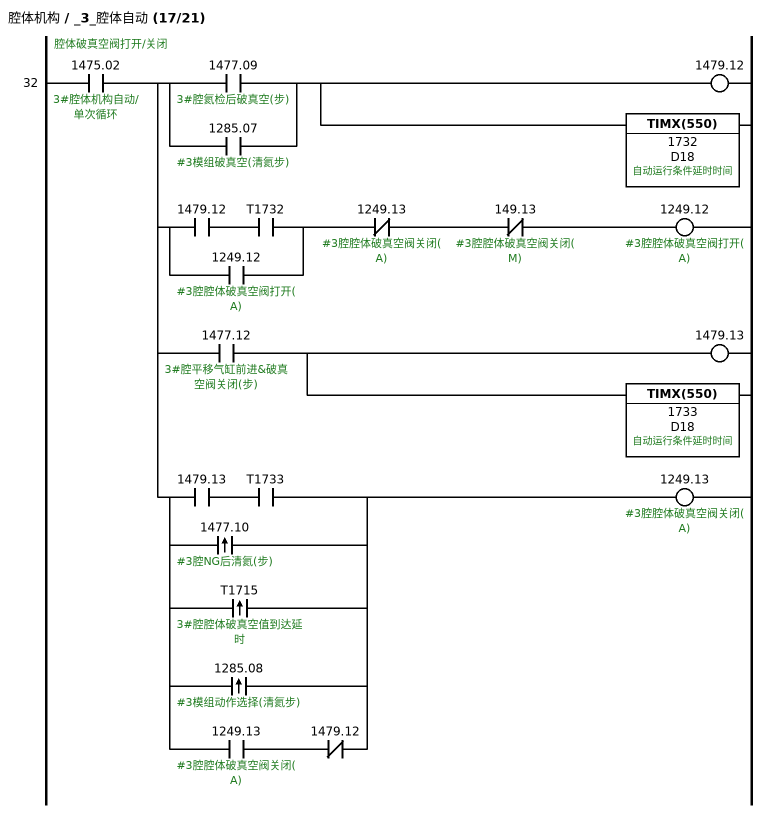
; [picture p336: 腔体机构 / _3_腔体自动, rungs 32-32]
; rung 32: 腔体破真空阀打开/关闭
LD 1475.02  ; 3#腔体机构自动/单次循环
OUT TR0
LD 1477.09  ; 3#腔氦检后破真空(步)
OR 1285.07  ; #3模组破真空(清氦步)
ANDLD
OUT 1479.12
TIMX(550) 1732 D18  ; 自动运行条件延时时间
LD TR0
LD 1479.12
AND T1732
OR 1249.12  ; #3腔腔体破真空阀打开(A)
ANDLD
ANDNOT 1249.13  ; #3腔腔体破真空阀关闭(A)
ANDNOT 149.13  ; #3腔腔体破真空阀关闭(M)
OUT 1249.12  ; #3腔腔体破真空阀打开(A)
LD TR0
AND 1477.12  ; 3#腔平移气缸前进&破真空阀关闭(步)
OUT 1479.13
TIMX(550) 1733 D18  ; 自动运行条件延时时间
LD TR0
LD 1479.13
AND T1733
@OR 1477.10  ; #3腔NG后清氦(步)
@OR T1715  ; 3#腔腔体破真空值到达延时
@OR 1285.08  ; #3模组动作选择(清氦步)
LD 1249.13  ; #3腔腔体破真空阀关闭(A)
ANDNOT 1479.12
ORLD
ANDLD
OUT 1249.13  ; #3腔腔体破真空阀关闭(A)

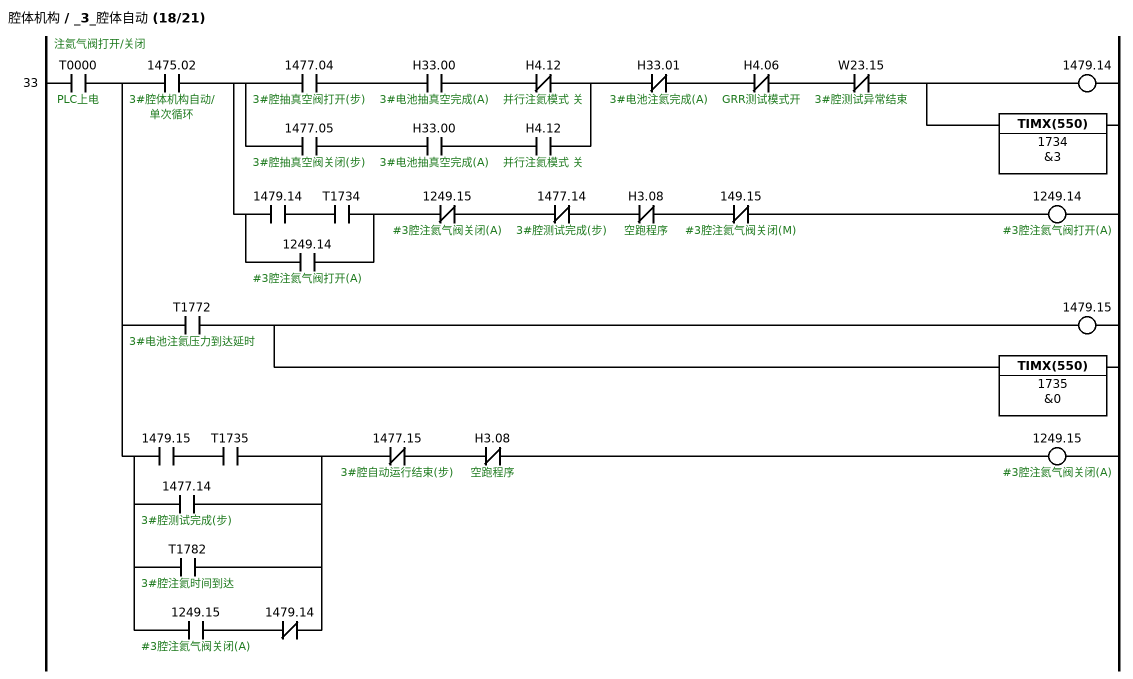
; rung 33: 注氦气阀打开/关闭
LD T0000  ; PLC上电
OUT TR0
AND 1475.02  ; 3#腔体机构自动/单次循环
OUT TR1
LD 1477.04  ; 3#腔抽真空阀打开(步)
AND H33.00  ; 3#电池抽真空完成(A)
ANDNOT H4.12  ; 并行注氦模式 关
LD 1477.05  ; 3#腔抽真空阀关闭(步)
AND H33.00  ; 3#电池抽真空完成(A)
AND H4.12  ; 并行注氦模式 关
ORLD
ANDLD
ANDNOT H33.01  ; 3#电池注氦完成(A)
ANDNOT H4.06  ; GRR测试模式开
ANDNOT W23.15  ; 3#腔测试异常结束
OUT 1479.14
TIMX(550) 1734 &3
LD TR1
LD 1479.14
AND T1734
OR 1249.14  ; #3腔注氦气阀打开(A)
ANDLD
ANDNOT 1249.15  ; #3腔注氦气阀关闭(A)
ANDNOT 1477.14  ; 3#腔测试完成(步)
ANDNOT H3.08  ; 空跑程序
ANDNOT 149.15  ; #3腔注氦气阀关闭(M)
OUT 1249.14  ; #3腔注氦气阀打开(A)
LD TR0
AND T1772  ; 3#电池注氦压力到达延时
OUT 1479.15
TIMX(550) 1735 &0
LD TR0
LD 1479.15
AND T1735
OR 1477.14  ; 3#腔测试完成(步)
OR T1782  ; 3#腔注氦时间到达
LD 1249.15  ; #3腔注氦气阀关闭(A)
ANDNOT 1479.14
ORLD
ANDLD
ANDNOT 1477.15  ; 3#腔自动运行结束(步)
ANDNOT H3.08  ; 空跑程序
OUT 1249.15  ; #3腔注氦气阀关闭(A)

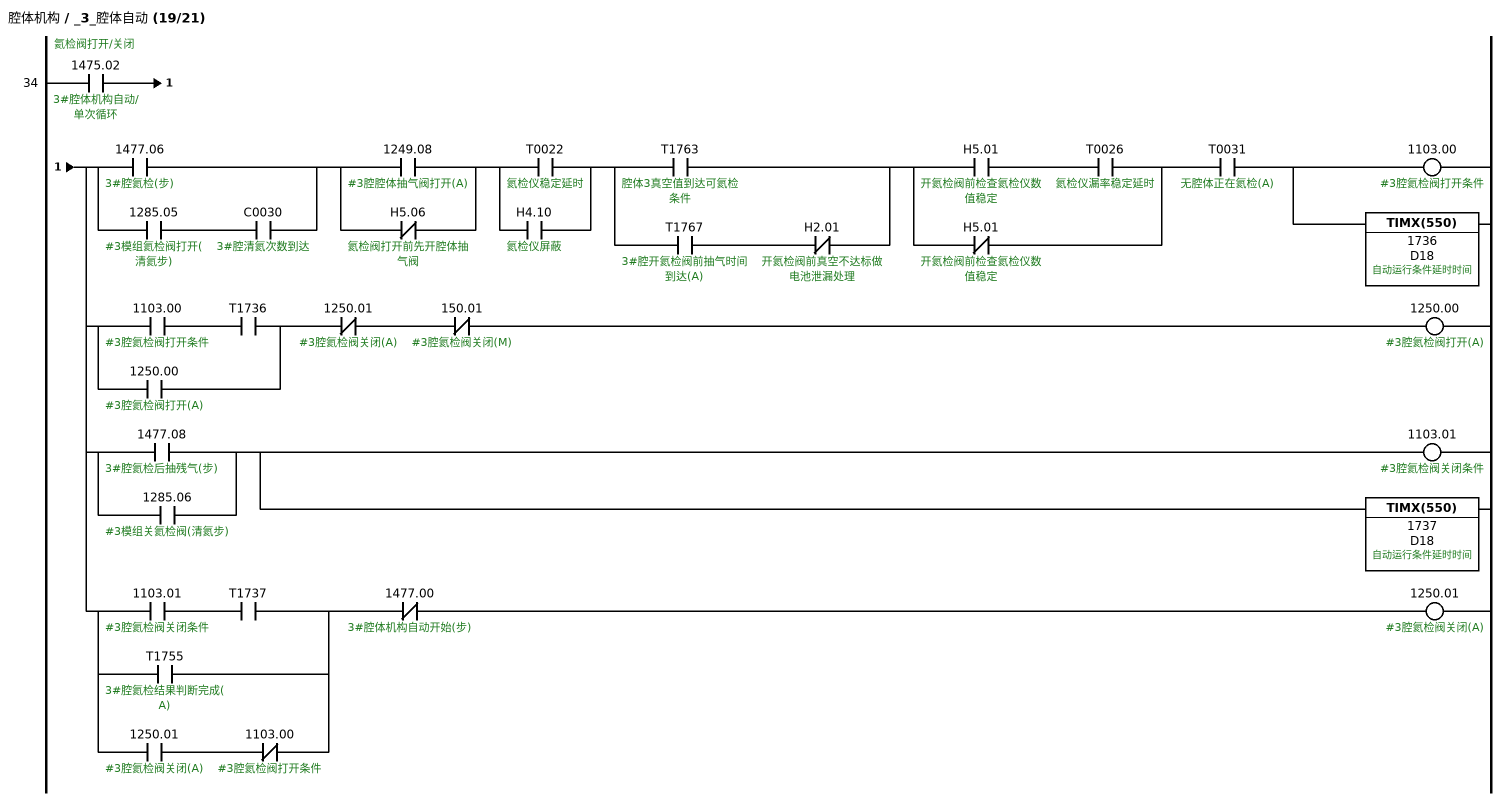
; rung 34: 氦检阀打开/关闭
LD 1475.02  ; 3#腔体机构自动/单次循环
OUT TR0
LD 1477.06  ; 3#腔氦检(步)
LD 1285.05  ; #3模组氦检阀打开(清氦步)
AND C0030  ; 3#腔清氦次数到达
ORLD
ANDLD
LD 1249.08  ; #3腔腔体抽气阀打开(A)
ORNOT H5.06  ; 氦检阀打开前先开腔体抽气阀
ANDLD
LD T0022  ; 氦检仪稳定延时
OR H4.10  ; 氦检仪屏蔽
ANDLD
LD T1763  ; 腔体3真空值到达可氦检条件
LD T1767  ; 3#腔开氦检阀前抽气时间到达(A)
ANDNOT H2.01  ; 开氦检阀前真空不达标做电池泄漏处理
ORLD
ANDLD
LD H5.01  ; 开氦检阀前检查氦检仪数值稳定
AND T0026  ; 氦检仪漏率稳定延时
ORNOT H5.01  ; 开氦检阀前检查氦检仪数值稳定
ANDLD
AND T0031  ; 无腔体正在氦检(A)
OUT 1103.00  ; #3腔氦检阀打开条件
TIMX(550) 1736 D18  ; 自动运行条件延时时间
LD TR0
LD 1103.00  ; #3腔氦检阀打开条件
AND T1736
OR 1250.00  ; #3腔氦检阀打开(A)
ANDLD
ANDNOT 1250.01  ; #3腔氦检阀关闭(A)
ANDNOT 150.01  ; #3腔氦检阀关闭(M)
OUT 1250.00  ; #3腔氦检阀打开(A)
LD TR0
LD 1477.08  ; 3#腔氦检后抽残气(步)
OR 1285.06  ; #3模组关氦检阀(清氦步)
ANDLD
OUT 1103.01  ; #3腔氦检阀关闭条件
TIMX(550) 1737 D18  ; 自动运行条件延时时间
LD TR0
LD 1103.01  ; #3腔氦检阀关闭条件
AND T1737
OR T1755  ; 3#腔氦检结果判断完成(A)
LD 1250.01  ; #3腔氦检阀关闭(A)
ANDNOT 1103.00  ; #3腔氦检阀打开条件
ORLD
ANDLD
ANDNOT 1477.00  ; 3#腔体机构自动开始(步)
OUT 1250.01  ; #3腔氦检阀关闭(A)

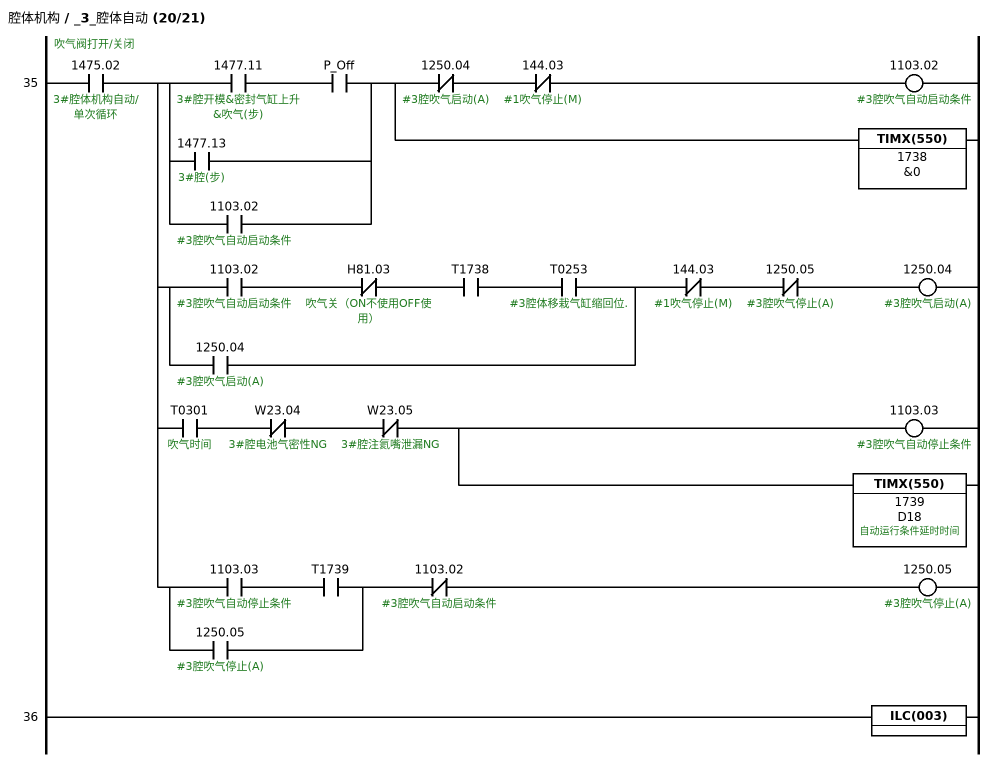
; rung 35: 吹气阀打开/关闭
LD 1475.02  ; 3#腔体机构自动/单次循环
OUT TR0
LD 1477.11  ; 3#腔开模&密封气缸上升&吹气(步)
AND P_Off
OR 1477.13  ; 3#腔(步)
OR 1103.02  ; #3腔吹气自动启动条件
ANDLD
OUT TR1
ANDNOT 1250.04  ; #3腔吹气启动(A)
ANDNOT 144.03  ; #1吹气停止(M)
OUT 1103.02  ; #3腔吹气自动启动条件
LD TR1
TIMX(550) 1738 &0
LD TR0
LD 1103.02  ; #3腔吹气自动启动条件
ANDNOT H81.03  ; 吹气关（ON不使用OFF使用）
AND T1738
AND T0253  ; #3腔体移栽气缸缩回位.
OR 1250.04  ; #3腔吹气启动(A)
ANDLD
ANDNOT 144.03  ; #1吹气停止(M)
ANDNOT 1250.05  ; #3腔吹气停止(A)
OUT 1250.04  ; #3腔吹气启动(A)
LD TR0
AND T0301  ; 吹气时间
ANDNOT W23.04  ; 3#腔电池气密性NG
ANDNOT W23.05  ; 3#腔注氦嘴泄漏NG
OUT 1103.03  ; #3腔吹气自动停止条件
TIMX(550) 1739 D18  ; 自动运行条件延时时间
LD TR0
LD 1103.03  ; #3腔吹气自动停止条件
AND T1739
OR 1250.05  ; #3腔吹气停止(A)
ANDLD
ANDNOT 1103.02  ; #3腔吹气自动启动条件
OUT 1250.05  ; #3腔吹气停止(A)
; rung 36
ILC(003)

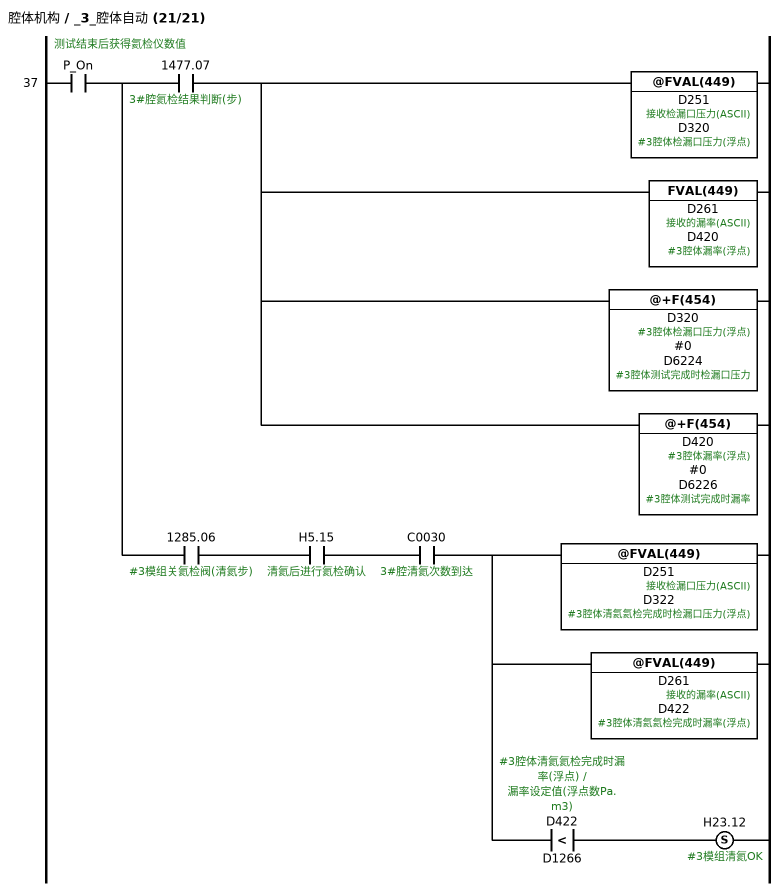
; rung 37: 测试结束后获得氦检仪数值
LD P_On
OUT TR0
AND 1477.07  ; 3#腔氦检结果判断(步)
@FVAL(449) D251 D320  ; 接收检漏口压力(ASCII), #3腔体检漏口压力(浮点)
FVAL(449) D261 D420  ; 接收的漏率(ASCII), #3腔体漏率(浮点)
@+F(454) D320 #0 D6224  ; #3腔体检漏口压力(浮点), #3腔体测试完成时检漏口压力
@+F(454) D420 #0 D6226  ; #3腔体漏率(浮点), #3腔体测试完成时漏率
LD TR0
AND 1285.06  ; #3模组关氦检阀(清氦步)
AND H5.15  ; 清氦后进行氦检确认
AND C0030  ; 3#腔清氦次数到达
@FVAL(449) D251 D322  ; 接收检漏口压力(ASCII), #3腔体清氦氦检完成时检漏口压力(浮点)
@FVAL(449) D261 D422  ; 接收的漏率(ASCII), #3腔体清氦氦检完成时漏率(浮点)
AND<F(331) D422 D1266  ; #3腔体清氦氦检完成时漏率(浮点), 漏率设定值(浮点数Pa.m3)
SET H23.12  ; #3模组清氦OK

### Section _4_腔体自动

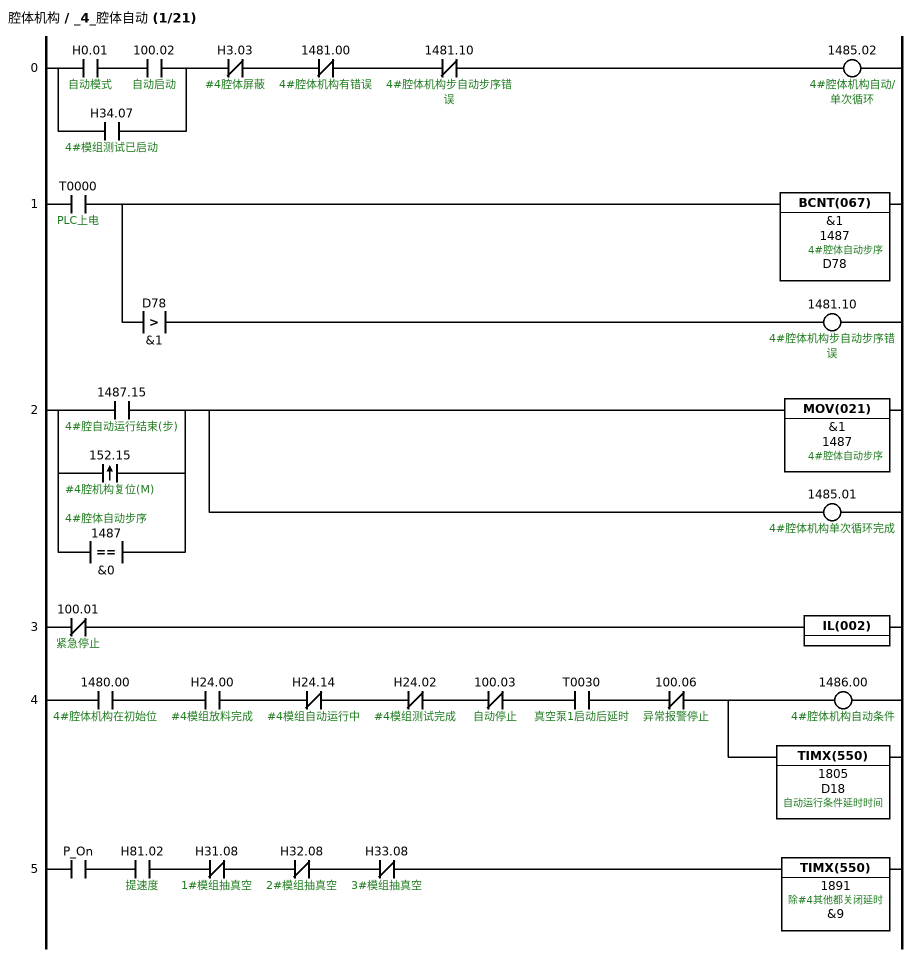
; rung 0
LD H0.01  ; 自动模式
AND 100.02  ; 自动启动
OR H34.07  ; 4#模组测试已启动
ANDNOT H3.03  ; #4腔体屏蔽
ANDNOT 1481.00  ; 4#腔体机构有错误
ANDNOT 1481.10  ; 4#腔体机构步自动步序错误
OUT 1485.02  ; 4#腔体机构自动/单次循环
; rung 1
LD T0000  ; PLC上电
BCNT(067) &1 1487 D78  ; 4#腔体自动步序
AND>(320) D78 &1
OUT 1481.10  ; 4#腔体机构步自动步序错误
; rung 2
LD 1487.15  ; 4#腔自动运行结束(步)
@OR 152.15  ; #4腔机构复位(M)
OR=(300) 1487 &0  ; 4#腔体自动步序
MOV(021) &1 1487  ; 4#腔体自动步序
OUT 1485.01  ; 4#腔体机构单次循环完成
; rung 3
LDNOT 100.01  ; 紧急停止
IL(002)
; rung 4
LD 1480.00  ; 4#腔体机构在初始位
AND H24.00  ; #4模组放料完成
ANDNOT H24.14  ; #4模组自动运行中
ANDNOT H24.02  ; #4模组测试完成
ANDNOT 100.03  ; 自动停止
AND T0030  ; 真空泵1启动后延时
ANDNOT 100.06  ; 异常报警停止
OUT 1486.00  ; 4#腔体机构自动条件
TIMX(550) 1805 D18  ; 自动运行条件延时时间
; rung 5
LD P_On
AND H81.02  ; 提速度
ANDNOT H31.08  ; 1#模组抽真空
ANDNOT H32.08  ; 2#模组抽真空
ANDNOT H33.08  ; 3#模组抽真空
TIMX(550) 1891 &9  ; 除#4其他都关闭延时

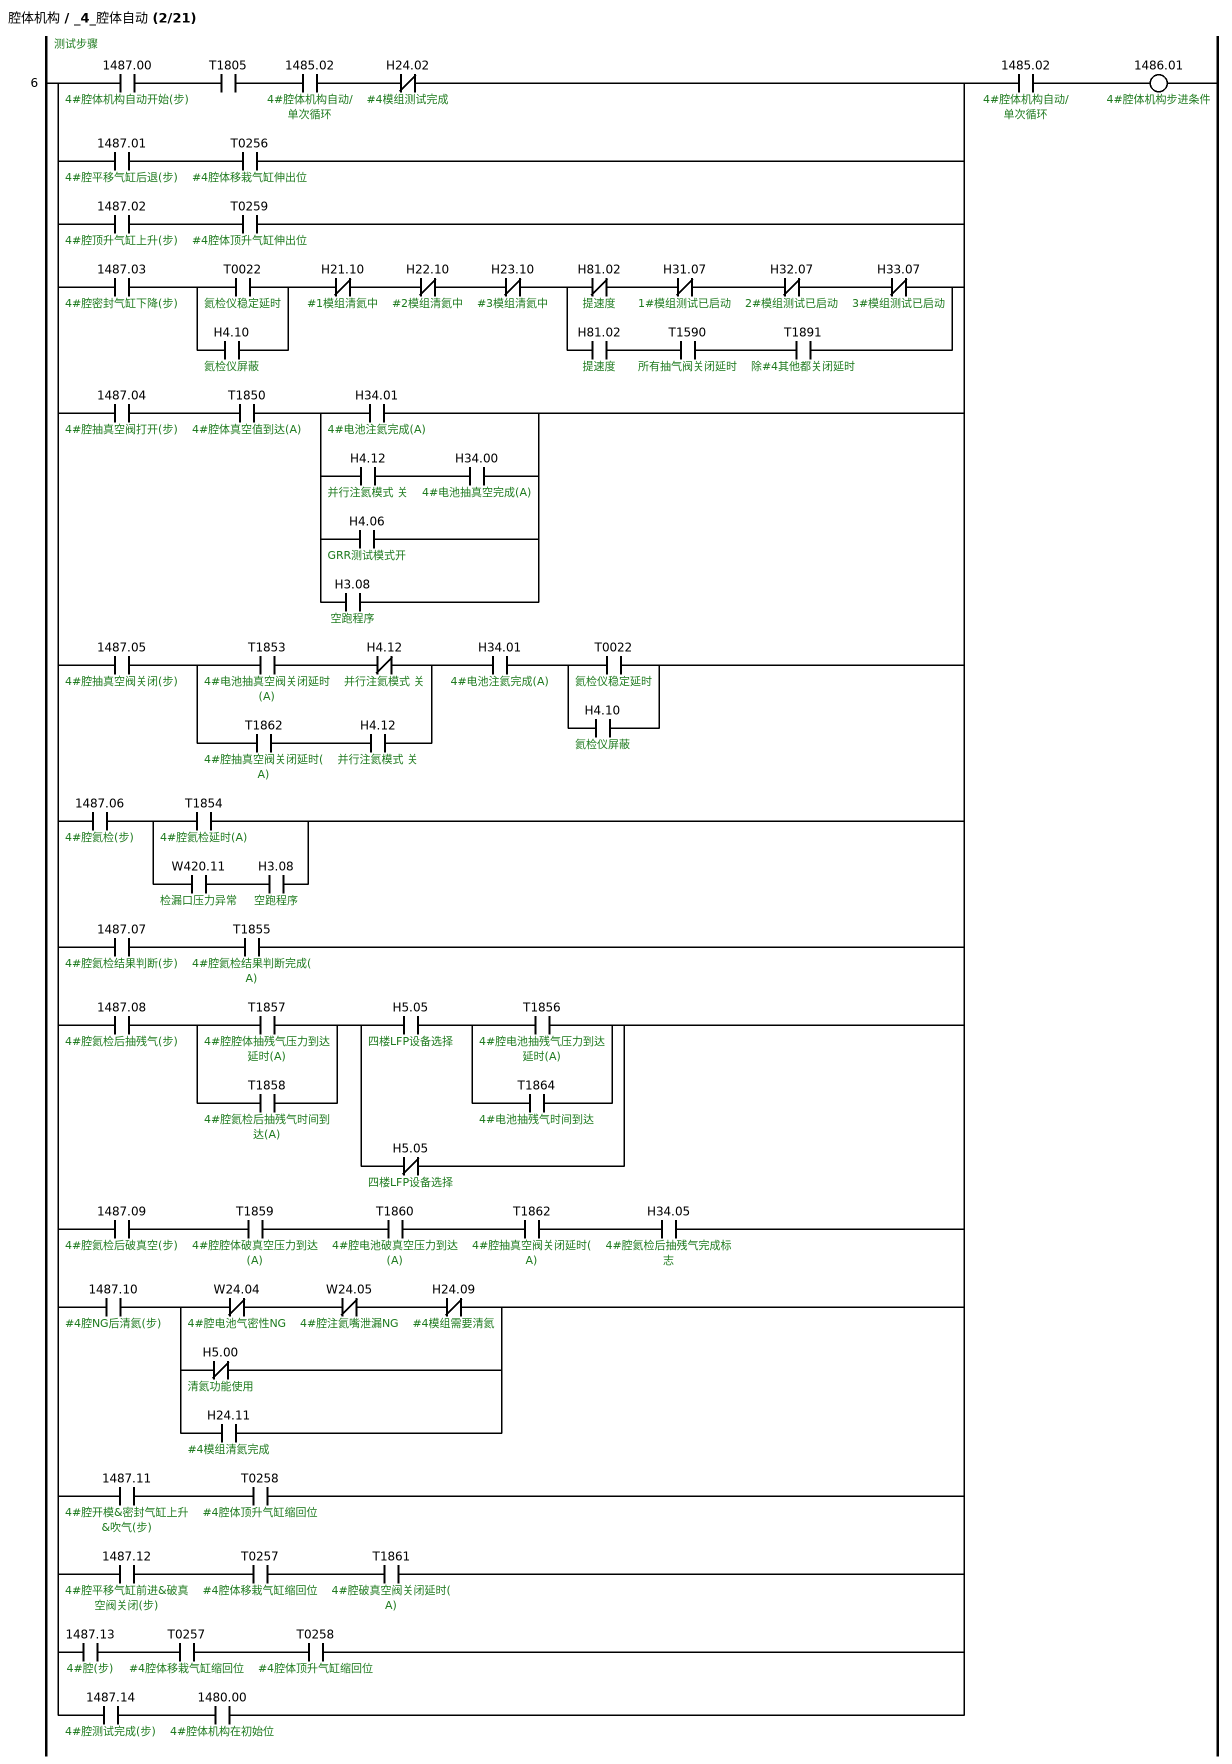
; rung 6: 测试步骤
LD 1487.00  ; 4#腔体机构自动开始(步)
AND T1805
AND 1485.02  ; 4#腔体机构自动/单次循环
ANDNOT H24.02  ; #4模组测试完成
LD 1487.01  ; 4#腔平移气缸后退(步)
AND T0256  ; #4腔体移栽气缸伸出位
ORLD
LD 1487.02  ; 4#腔顶升气缸上升(步)
AND T0259  ; #4腔体顶升气缸伸出位
ORLD
LD 1487.03  ; 4#腔密封气缸下降(步)
LD T0022  ; 氦检仪稳定延时
OR H4.10  ; 氦检仪屏蔽
ANDLD
ANDNOT H21.10  ; #1模组清氦中
ANDNOT H22.10  ; #2模组清氦中
ANDNOT H23.10  ; #3模组清氦中
LDNOT H81.02  ; 提速度
ANDNOT H31.07  ; 1#模组测试已启动
ANDNOT H32.07  ; 2#模组测试已启动
ANDNOT H33.07  ; 3#模组测试已启动
LD H81.02  ; 提速度
AND T1590  ; 所有抽气阀关闭延时
AND T1891  ; 除#4其他都关闭延时
ORLD
ANDLD
ORLD
LD 1487.04  ; 4#腔抽真空阀打开(步)
AND T1850  ; 4#腔体真空值到达(A)
LD H34.01  ; 4#电池注氦完成(A)
LD H4.12  ; 并行注氦模式 关
AND H34.00  ; 4#电池抽真空完成(A)
ORLD
OR H4.06  ; GRR测试模式开
OR H3.08  ; 空跑程序
ANDLD
ORLD
LD 1487.05  ; 4#腔抽真空阀关闭(步)
LD T1853  ; 4#电池抽真空阀关闭延时(A)
ANDNOT H4.12  ; 并行注氦模式 关
LD T1862  ; 4#腔抽真空阀关闭延时(A)
AND H4.12  ; 并行注氦模式 关
ORLD
ANDLD
AND H34.01  ; 4#电池注氦完成(A)
LD T0022  ; 氦检仪稳定延时
OR H4.10  ; 氦检仪屏蔽
ANDLD
ORLD
LD 1487.06  ; 4#腔氦检(步)
LD T1854  ; 4#腔氦检延时(A)
LD W420.11  ; 检漏口压力异常
AND H3.08  ; 空跑程序
ORLD
ANDLD
ORLD
LD 1487.07  ; 4#腔氦检结果判断(步)
AND T1855  ; 4#腔氦检结果判断完成(A)
ORLD
LD 1487.08  ; 4#腔氦检后抽残气(步)
LD T1857  ; 4#腔腔体抽残气压力到达延时(A)
OR T1858  ; 4#腔氦检后抽残气时间到达(A)
ANDLD
LD H5.05  ; 四楼LFP设备选择
LD T1856  ; 4#腔电池抽残气压力到达延时(A)
OR T1864  ; 4#电池抽残气时间到达
ANDLD
ORNOT H5.05  ; 四楼LFP设备选择
ANDLD
ORLD
LD 1487.09  ; 4#腔氦检后破真空(步)
AND T1859  ; 4#腔腔体破真空压力到达(A)
AND T1860  ; 4#腔电池破真空压力到达(A)
AND T1862  ; 4#腔抽真空阀关闭延时(A)
AND H34.05  ; 4#腔氦检后抽残气完成标志
ORLD
LD 1487.10  ; #4腔NG后清氦(步)
LDNOT W24.04  ; 4#腔电池气密性NG
ANDNOT W24.05  ; 4#腔注氦嘴泄漏NG
ANDNOT H24.09  ; #4模组需要清氦
ORNOT H5.00  ; 清氦功能使用
OR H24.11  ; #4模组清氦完成
ANDLD
ORLD
LD 1487.11  ; 4#腔开模&密封气缸上升&吹气(步)
AND T0258  ; #4腔体顶升气缸缩回位
ORLD
LD 1487.12  ; 4#腔平移气缸前进&破真空阀关闭(步)
AND T0257  ; #4腔体移栽气缸缩回位
AND T1861  ; 4#腔破真空阀关闭延时(A)
ORLD
LD 1487.13  ; 4#腔(步)
AND T0257  ; #4腔体移栽气缸缩回位
AND T0258  ; #4腔体顶升气缸缩回位
ORLD
LD 1487.14  ; 4#腔测试完成(步)
AND 1480.00  ; 4#腔体机构在初始位
ORLD
AND 1485.02  ; 4#腔体机构自动/单次循环
OUT 1486.01  ; 4#腔体机构步进条件

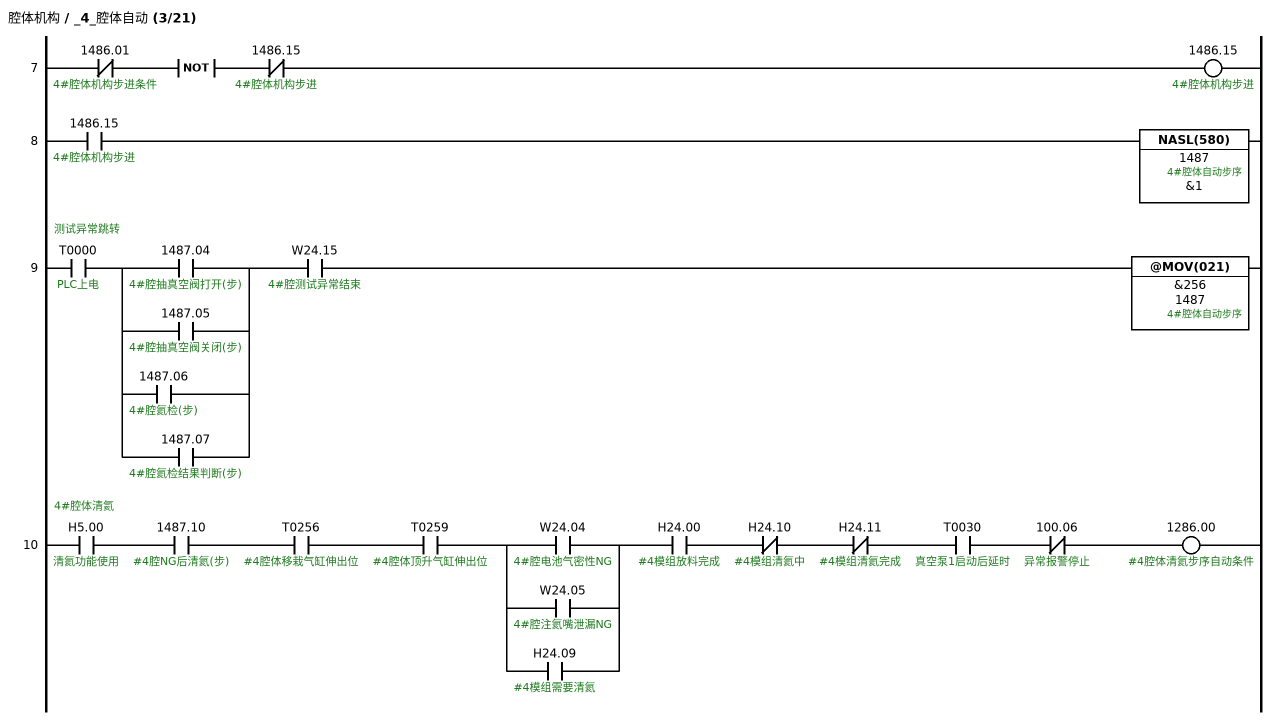
; rung 7
LDNOT 1486.01  ; 4#腔体机构步进条件
NOT(520)
ANDNOT 1486.15  ; 4#腔体机构步进
OUT 1486.15  ; 4#腔体机构步进
; rung 8
LD 1486.15  ; 4#腔体机构步进
NASL(580) 1487 &1  ; 4#腔体自动步序
; rung 9: 测试异常跳转
LD T0000  ; PLC上电
LD 1487.04  ; 4#腔抽真空阀打开(步)
OR 1487.05  ; 4#腔抽真空阀关闭(步)
OR 1487.06  ; 4#腔氦检(步)
OR 1487.07  ; 4#腔氦检结果判断(步)
ANDLD
AND W24.15  ; 4#腔测试异常结束
@MOV(021) &256 1487  ; 4#腔体自动步序
; rung 10: 4#腔体清氦
LD H5.00  ; 清氦功能使用
AND 1487.10  ; #4腔NG后清氦(步)
AND T0256  ; #4腔体移栽气缸伸出位
AND T0259  ; #4腔体顶升气缸伸出位
LD W24.04  ; 4#腔电池气密性NG
OR W24.05  ; 4#腔注氦嘴泄漏NG
OR H24.09  ; #4模组需要清氦
ANDLD
AND H24.00  ; #4模组放料完成
ANDNOT H24.10  ; #4模组清氦中
ANDNOT H24.11  ; #4模组清氦完成
AND T0030  ; 真空泵1启动后延时
ANDNOT 100.06  ; 异常报警停止
OUT 1286.00  ; #4腔体清氦步序自动条件

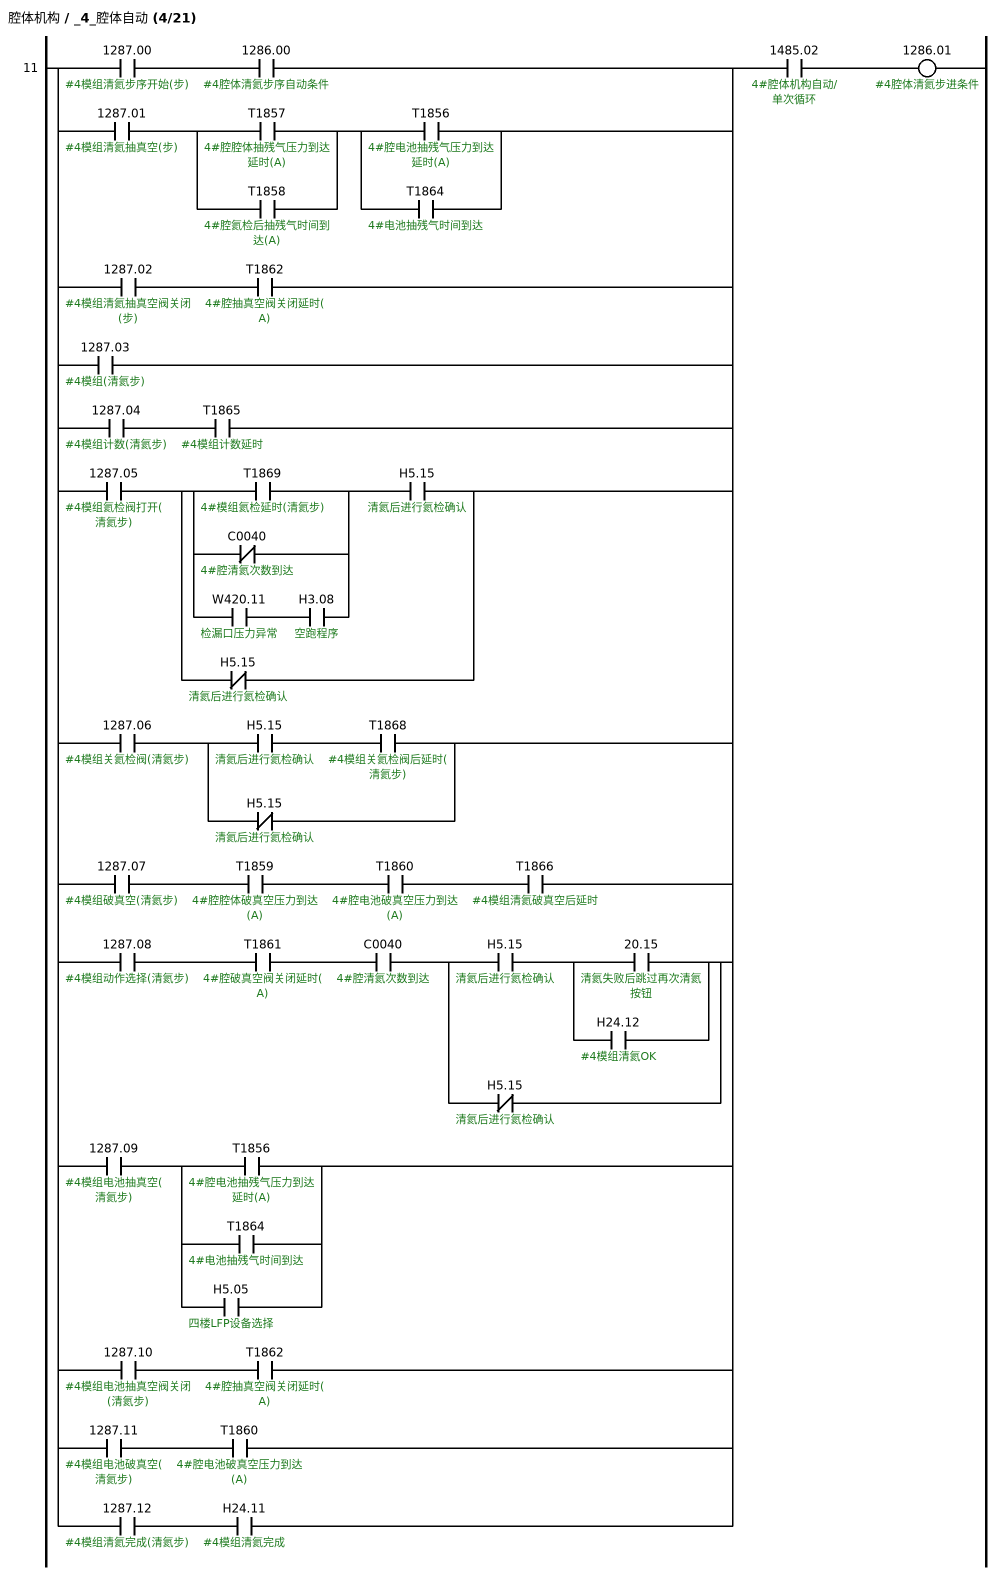
; rung 11
LD 1287.00  ; #4模组清氦步序开始(步)
AND 1286.00  ; #4腔体清氦步序自动条件
LD 1287.01  ; #4模组清氦抽真空(步)
LD T1857  ; 4#腔腔体抽残气压力到达延时(A)
OR T1858  ; 4#腔氦检后抽残气时间到达(A)
ANDLD
LD T1856  ; 4#腔电池抽残气压力到达延时(A)
OR T1864  ; 4#电池抽残气时间到达
ANDLD
ORLD
LD 1287.02  ; #4模组清氦抽真空阀关闭(步)
AND T1862  ; 4#腔抽真空阀关闭延时(A)
ORLD
OR 1287.03  ; #4模组(清氦步)
LD 1287.04  ; #4模组计数(清氦步)
AND T1865  ; #4模组计数延时
ORLD
LD 1287.05  ; #4模组氦检阀打开(清氦步)
LD T1869  ; 4#模组氦检延时(清氦步)
ORNOT C0040  ; 4#腔清氦次数到达
LD W420.11  ; 检漏口压力异常
AND H3.08  ; 空跑程序
ORLD
AND H5.15  ; 清氦后进行氦检确认
ORNOT H5.15  ; 清氦后进行氦检确认
ANDLD
ORLD
LD 1287.06  ; #4模组关氦检阀(清氦步)
LD H5.15  ; 清氦后进行氦检确认
AND T1868  ; #4模组关氦检阀后延时(清氦步)
ORNOT H5.15  ; 清氦后进行氦检确认
ANDLD
ORLD
LD 1287.07  ; #4模组破真空(清氦步)
AND T1859  ; 4#腔腔体破真空压力到达(A)
AND T1860  ; 4#腔电池破真空压力到达(A)
AND T1866  ; #4模组清氦破真空后延时
ORLD
LD 1287.08  ; #4模组动作选择(清氦步)
AND T1861  ; 4#腔破真空阀关闭延时(A)
AND C0040  ; 4#腔清氦次数到达
LD H5.15  ; 清氦后进行氦检确认
LD 20.15  ; 清氦失败后跳过再次清氦按钮
OR H24.12  ; #4模组清氦OK
ANDLD
ORNOT H5.15  ; 清氦后进行氦检确认
ANDLD
ORLD
LD 1287.09  ; #4模组电池抽真空(清氦步)
LD T1856  ; 4#腔电池抽残气压力到达延时(A)
OR T1864  ; 4#电池抽残气时间到达
OR H5.05  ; 四楼LFP设备选择
ANDLD
ORLD
LD 1287.10  ; #4模组电池抽真空阀关闭(清氦步)
AND T1862  ; 4#腔抽真空阀关闭延时(A)
ORLD
LD 1287.11  ; #4模组电池破真空(清氦步)
AND T1860  ; 4#腔电池破真空压力到达(A)
ORLD
LD 1287.12  ; #4模组清氦完成(清氦步)
AND H24.11  ; #4模组清氦完成
ORLD
AND 1485.02  ; 4#腔体机构自动/单次循环
OUT 1286.01  ; #4腔体清氦步进条件

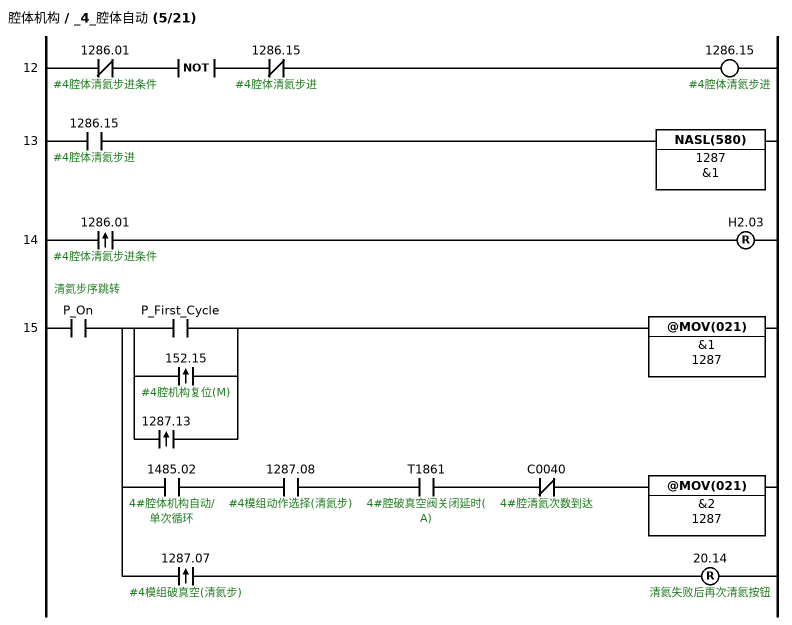
; rung 12
LDNOT 1286.01  ; #4腔体清氦步进条件
NOT(520)
ANDNOT 1286.15  ; #4腔体清氦步进
OUT 1286.15  ; #4腔体清氦步进
; rung 13
LD 1286.15  ; #4腔体清氦步进
NASL(580) 1287 &1
; rung 14
@LD 1286.01  ; #4腔体清氦步进条件
RSET H2.03
; rung 15: 清氦步序跳转
LD P_On
OUT TR0
LD P_First_Cycle
@OR 152.15  ; #4腔机构复位(M)
@OR 1287.13
ANDLD
@MOV(021) &1 1287
LD TR0
AND 1485.02  ; 4#腔体机构自动/单次循环
AND 1287.08  ; #4模组动作选择(清氦步)
AND T1861  ; 4#腔破真空阀关闭延时(A)
ANDNOT C0040  ; 4#腔清氦次数到达
@MOV(021) &2 1287
LD TR0
@AND 1287.07  ; #4模组破真空(清氦步)
RSET 20.14  ; 清氦失败后再次清氦按钮

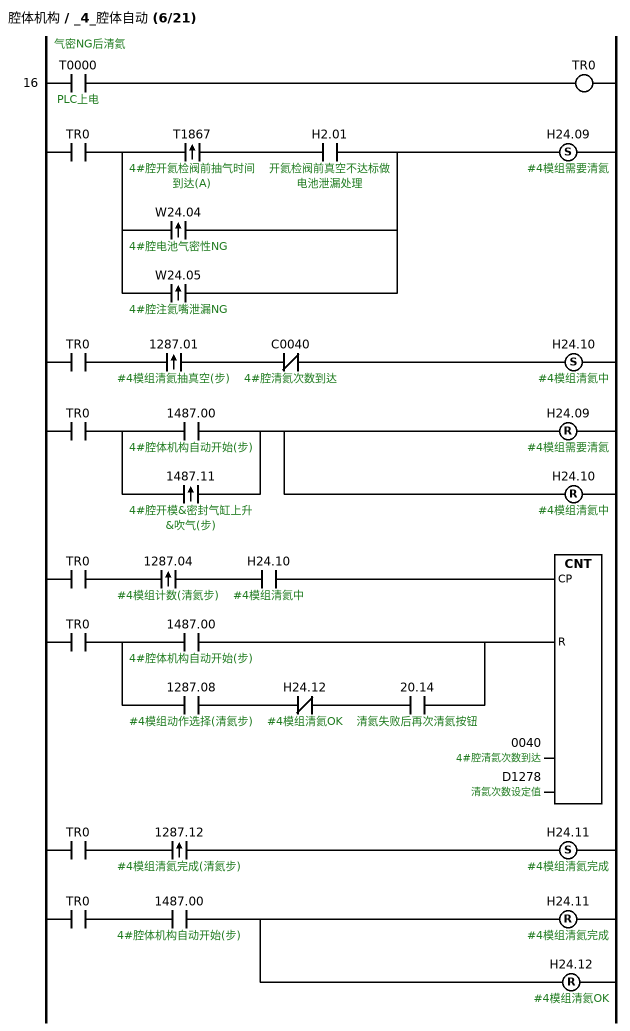
; rung 16: 气密NG后清氦
LD T0000  ; PLC上电
OUT TR0
@LD T1867  ; 4#腔开氦检阀前抽气时间到达(A)
AND H2.01  ; 开氦检阀前真空不达标做电池泄漏处理
@OR W24.04  ; 4#腔电池气密性NG
@OR W24.05  ; 4#腔注氦嘴泄漏NG
ANDLD
SET H24.09  ; #4模组需要清氦
LD TR0
@AND 1287.01  ; #4模组清氦抽真空(步)
ANDNOT C0040  ; 4#腔清氦次数到达
SET H24.10  ; #4模组清氦中
LD TR0
LD 1487.00  ; 4#腔体机构自动开始(步)
@OR 1487.11  ; 4#腔开模&密封气缸上升&吹气(步)
ANDLD
RSET H24.09  ; #4模组需要清氦
RSET H24.10  ; #4模组清氦中
LD TR0
@AND 1287.04  ; #4模组计数(清氦步)
AND H24.10  ; #4模组清氦中
LD TR0
LD 1487.00  ; 4#腔体机构自动开始(步)
LD 1287.08  ; #4模组动作选择(清氦步)
ANDNOT H24.12  ; #4模组清氦OK
AND 20.14  ; 清氦失败后再次清氦按钮
ORLD
ANDLD
CNT 0040 D1278  ; 清氦次数设定值, 4#腔清氦次数到达
LD TR0
@AND 1287.12  ; #4模组清氦完成(清氦步)
SET H24.11  ; #4模组清氦完成
LD TR0
AND 1487.00  ; 4#腔体机构自动开始(步)
RSET H24.11  ; #4模组清氦完成
RSET H24.12  ; #4模组清氦OK

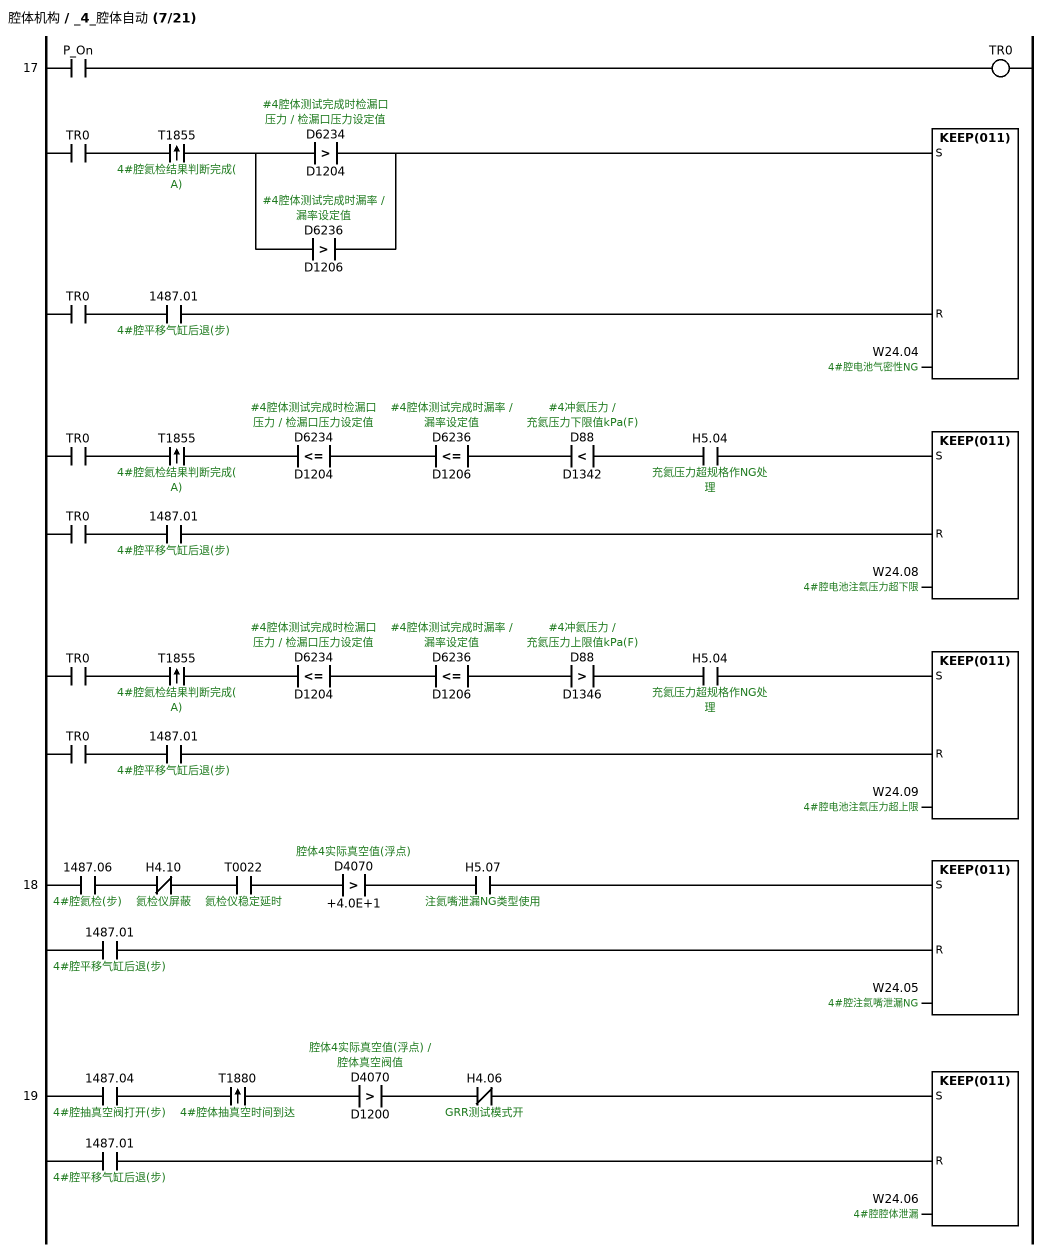
; rung 17
LD P_On
OUT TR0
@AND T1855  ; 4#腔氦检结果判断完成(A)
LD>F(333) D6234 D1204  ; #4腔体测试完成时检漏口压力, 检漏口压力设定值
OR>F(333) D6236 D1206  ; #4腔体测试完成时漏率, 漏率设定值
ANDLD
LD TR0
AND 1487.01  ; 4#腔平移气缸后退(步)
KEEP(011) W24.04  ; 4#腔电池气密性NG
LD TR0
@AND T1855  ; 4#腔氦检结果判断完成(A)
AND<=F(332) D6234 D1204  ; #4腔体测试完成时检漏口压力, 检漏口压力设定值
AND<=F(332) D6236 D1206  ; #4腔体测试完成时漏率, 漏率设定值
AND<F(331) D88 D1342  ; #4冲氦压力, 充氦压力下限值kPa(F)
AND H5.04  ; 充氦压力超规格作NG处理
LD TR0
AND 1487.01  ; 4#腔平移气缸后退(步)
KEEP(011) W24.08  ; 4#腔电池注氦压力超下限
LD TR0
@AND T1855  ; 4#腔氦检结果判断完成(A)
AND<=F(332) D6234 D1204  ; #4腔体测试完成时检漏口压力, 检漏口压力设定值
AND<=F(332) D6236 D1206  ; #4腔体测试完成时漏率, 漏率设定值
AND>F(333) D88 D1346  ; #4冲氦压力, 充氦压力上限值kPa(F)
AND H5.04  ; 充氦压力超规格作NG处理
LD TR0
AND 1487.01  ; 4#腔平移气缸后退(步)
KEEP(011) W24.09  ; 4#腔电池注氦压力超上限
; rung 18
LD 1487.06  ; 4#腔氦检(步)
ANDNOT H4.10  ; 氦检仪屏蔽
AND T0022  ; 氦检仪稳定延时
AND>F(333) D4070 +4.0E+1  ; 腔体4实际真空值(浮点)
AND H5.07  ; 注氦嘴泄漏NG类型使用
LD 1487.01  ; 4#腔平移气缸后退(步)
KEEP(011) W24.05  ; 4#腔注氦嘴泄漏NG
; rung 19
LD 1487.04  ; 4#腔抽真空阀打开(步)
@AND T1880  ; 4#腔体抽真空时间到达
AND>F(333) D4070 D1200  ; 腔体4实际真空值(浮点), 腔体真空阀值
ANDNOT H4.06  ; GRR测试模式开
LD 1487.01  ; 4#腔平移气缸后退(步)
KEEP(011) W24.06  ; 4#腔腔体泄漏

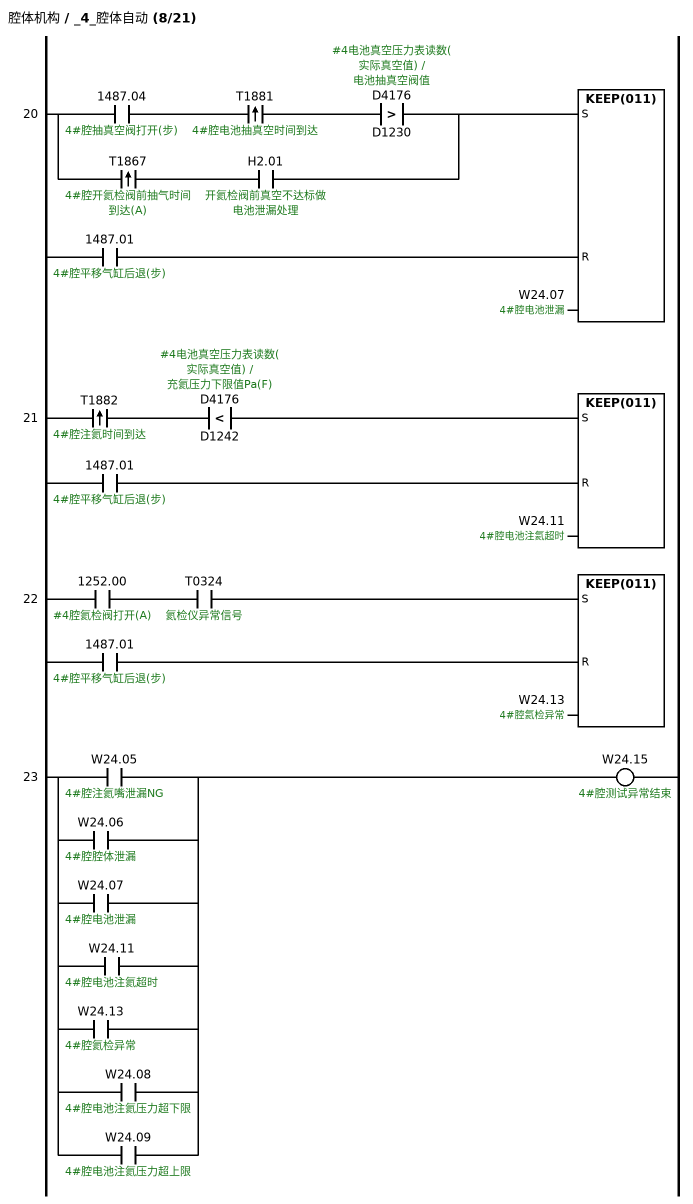
; rung 20
LD 1487.04  ; 4#腔抽真空阀打开(步)
@AND T1881  ; 4#腔电池抽真空时间到达
AND>F(333) D4176 D1230  ; #4电池真空压力表读数(实际真空值), 电池抽真空阀值
@LD T1867  ; 4#腔开氦检阀前抽气时间到达(A)
AND H2.01  ; 开氦检阀前真空不达标做电池泄漏处理
ORLD
LD 1487.01  ; 4#腔平移气缸后退(步)
KEEP(011) W24.07  ; 4#腔电池泄漏
; rung 21
@LD T1882  ; 4#腔注氦时间到达
AND<F(331) D4176 D1242  ; #4电池真空压力表读数(实际真空值), 充氦压力下限值Pa(F)
LD 1487.01  ; 4#腔平移气缸后退(步)
KEEP(011) W24.11  ; 4#腔电池注氦超时
; rung 22
LD 1252.00  ; #4腔氦检阀打开(A)
AND T0324  ; 氦检仪异常信号
LD 1487.01  ; 4#腔平移气缸后退(步)
KEEP(011) W24.13  ; 4#腔氦检异常
; rung 23
LD W24.05  ; 4#腔注氦嘴泄漏NG
OR W24.06  ; 4#腔腔体泄漏
OR W24.07  ; 4#腔电池泄漏
OR W24.11  ; 4#腔电池注氦超时
OR W24.13  ; 4#腔氦检异常
OR W24.08  ; 4#腔电池注氦压力超下限
OR W24.09  ; 4#腔电池注氦压力超上限
OUT W24.15  ; 4#腔测试异常结束

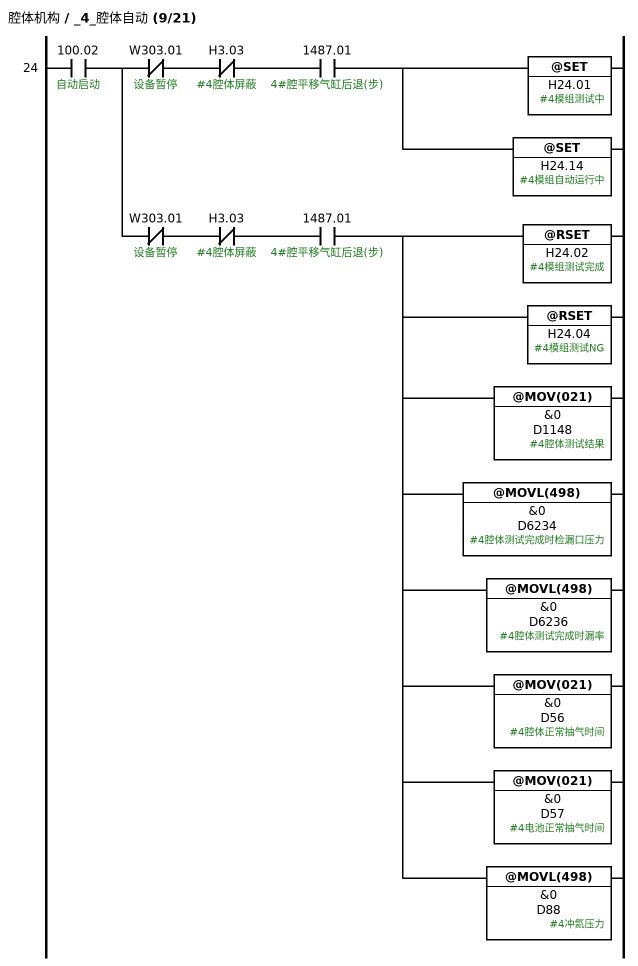
; rung 24
LD 100.02  ; 自动启动
OUT TR0
ANDNOT W303.01  ; 设备暂停
ANDNOT H3.03  ; #4腔体屏蔽
AND 1487.01  ; 4#腔平移气缸后退(步)
@SET H24.01  ; #4模组测试中
@SET H24.14  ; #4模组自动运行中
LD TR0
ANDNOT W303.01  ; 设备暂停
ANDNOT H3.03  ; #4腔体屏蔽
AND 1487.01  ; 4#腔平移气缸后退(步)
@RSET H24.02  ; #4模组测试完成
@RSET H24.04  ; #4模组测试NG
@MOV(021) &0 D1148  ; #4腔体测试结果
@MOVL(498) &0 D6234  ; #4腔体测试完成时检漏口压力
@MOVL(498) &0 D6236  ; #4腔体测试完成时漏率
@MOV(021) &0 D56  ; #4腔体正常抽气时间
@MOV(021) &0 D57  ; #4电池正常抽气时间
@MOVL(498) &0 D88  ; #4冲氦压力

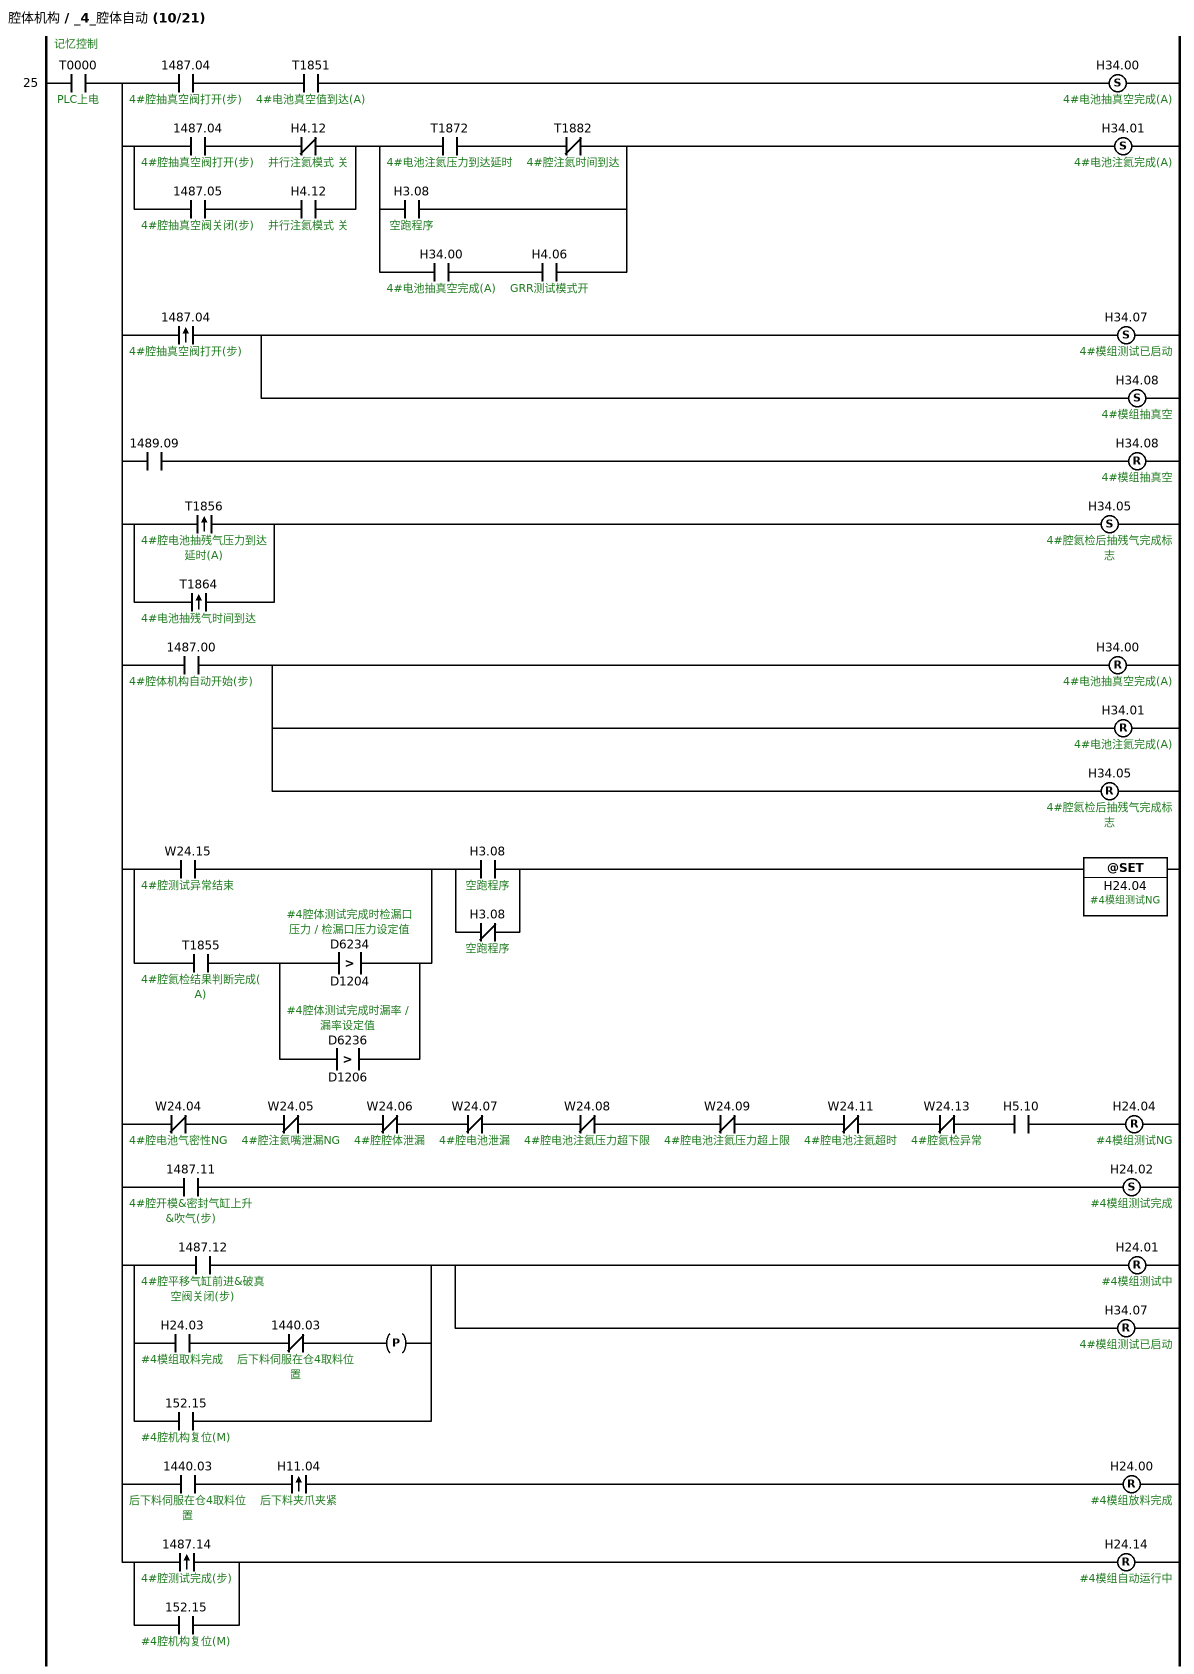
; rung 25: 记忆控制
LD T0000  ; PLC上电
OUT TR0
AND 1487.04  ; 4#腔抽真空阀打开(步)
AND T1851  ; 4#电池真空值到达(A)
SET H34.00  ; 4#电池抽真空完成(A)
LD TR0
LD 1487.04  ; 4#腔抽真空阀打开(步)
ANDNOT H4.12  ; 并行注氦模式 关
LD 1487.05  ; 4#腔抽真空阀关闭(步)
AND H4.12  ; 并行注氦模式 关
ORLD
ANDLD
LD T1872  ; 4#电池注氦压力到达延时
ANDNOT T1882  ; 4#腔注氦时间到达
OR H3.08  ; 空跑程序
LD H34.00  ; 4#电池抽真空完成(A)
AND H4.06  ; GRR测试模式开
ORLD
ANDLD
SET H34.01  ; 4#电池注氦完成(A)
LD TR0
@AND 1487.04  ; 4#腔抽真空阀打开(步)
SET H34.07  ; 4#模组测试已启动
SET H34.08  ; 4#模组抽真空
LD TR0
AND 1489.09
RSET H34.08  ; 4#模组抽真空
LD TR0
@LD T1856  ; 4#腔电池抽残气压力到达延时(A)
@OR T1864  ; 4#电池抽残气时间到达
ANDLD
SET H34.05  ; 4#腔氦检后抽残气完成标志
LD TR0
AND 1487.00  ; 4#腔体机构自动开始(步)
RSET H34.00  ; 4#电池抽真空完成(A)
RSET H34.01  ; 4#电池注氦完成(A)
RSET H34.05  ; 4#腔氦检后抽残气完成标志
LD TR0
LD W24.15  ; 4#腔测试异常结束
LD T1855  ; 4#腔氦检结果判断完成(A)
LD>F(333) D6234 D1204  ; #4腔体测试完成时检漏口压力, 检漏口压力设定值
OR>F(333) D6236 D1206  ; #4腔体测试完成时漏率, 漏率设定值
ANDLD
ORLD
ANDLD
LD H3.08  ; 空跑程序
ORNOT H3.08  ; 空跑程序
ANDLD
@SET H24.04  ; #4模组测试NG
LD TR0
ANDNOT W24.04  ; 4#腔电池气密性NG
ANDNOT W24.05  ; 4#腔注氦嘴泄漏NG
ANDNOT W24.06  ; 4#腔腔体泄漏
ANDNOT W24.07  ; 4#腔电池泄漏
ANDNOT W24.08  ; 4#腔电池注氦压力超下限
ANDNOT W24.09  ; 4#腔电池注氦压力超上限
ANDNOT W24.11  ; 4#腔电池注氦超时
ANDNOT W24.13  ; 4#腔氦检异常
AND H5.10
RSET H24.04  ; #4模组测试NG
LD TR0
AND 1487.11  ; 4#腔开模&密封气缸上升&吹气(步)
SET H24.02  ; #4模组测试完成
LD TR0
LD 1487.12  ; 4#腔平移气缸前进&破真空阀关闭(步)
LD H24.03  ; #4模组取料完成
ANDNOT 1440.03  ; 后下料伺服在仓4取料位置
UP(521)
ORLD
OR 152.15  ; #4腔机构复位(M)
ANDLD
RSET H24.01  ; #4模组测试中
RSET H34.07  ; 4#模组测试已启动
LD TR0
AND 1440.03  ; 后下料伺服在仓4取料位置
@AND H11.04  ; 后下料夹爪夹紧
RSET H24.00  ; #4模组放料完成
LD TR0
@LD 1487.14  ; 4#腔测试完成(步)
OR 152.15  ; #4腔机构复位(M)
ANDLD
RSET H24.14  ; #4模组自动运行中

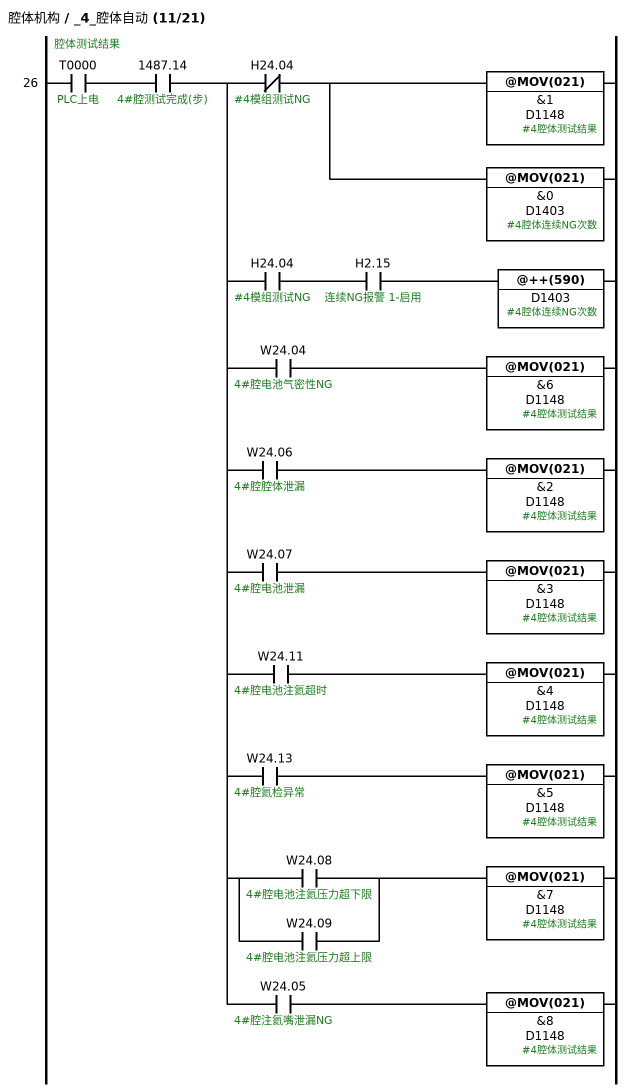
; rung 26: 腔体测试结果
LD T0000  ; PLC上电
AND 1487.14  ; 4#腔测试完成(步)
OUT TR0
ANDNOT H24.04  ; #4模组测试NG
@MOV(021) &1 D1148  ; #4腔体测试结果
@MOV(021) &0 D1403  ; #4腔体连续NG次数
LD TR0
AND H24.04  ; #4模组测试NG
AND H2.15  ; 连续NG报警 1-启用
@++(590) D1403  ; #4腔体连续NG次数
LD TR0
AND W24.04  ; 4#腔电池气密性NG
@MOV(021) &6 D1148  ; #4腔体测试结果
LD TR0
AND W24.06  ; 4#腔腔体泄漏
@MOV(021) &2 D1148  ; #4腔体测试结果
LD TR0
AND W24.07  ; 4#腔电池泄漏
@MOV(021) &3 D1148  ; #4腔体测试结果
LD TR0
AND W24.11  ; 4#腔电池注氦超时
@MOV(021) &4 D1148  ; #4腔体测试结果
LD TR0
AND W24.13  ; 4#腔氦检异常
@MOV(021) &5 D1148  ; #4腔体测试结果
LD TR0
LD W24.08  ; 4#腔电池注氦压力超下限
OR W24.09  ; 4#腔电池注氦压力超上限
ANDLD
@MOV(021) &7 D1148  ; #4腔体测试结果
LD TR0
AND W24.05  ; 4#腔注氦嘴泄漏NG
@MOV(021) &8 D1148  ; #4腔体测试结果

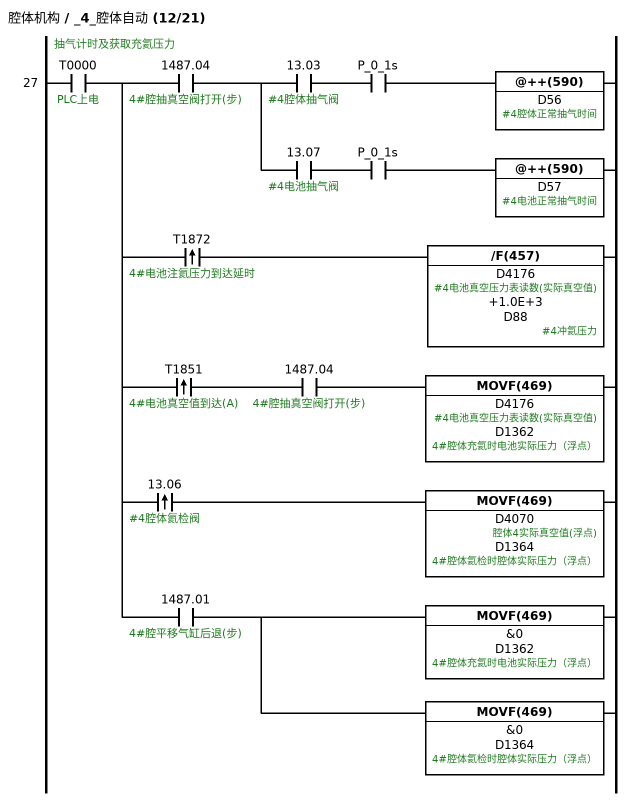
; rung 27: 抽气计时及获取充氦压力
LD T0000  ; PLC上电
OUT TR0
AND 1487.04  ; 4#腔抽真空阀打开(步)
OUT TR1
AND 13.03  ; #4腔体抽气阀
AND P_0_1s
@++(590) D56  ; #4腔体正常抽气时间
LD TR1
AND 13.07  ; #4电池抽气阀
AND P_0_1s
@++(590) D57  ; #4电池正常抽气时间
LD TR0
@AND T1872  ; 4#电池注氦压力到达延时
/F(457) D4176 +1.0E+3 D88  ; #4电池真空压力表读数(实际真空值), #4冲氦压力
LD TR0
@AND T1851  ; 4#电池真空值到达(A)
AND 1487.04  ; 4#腔抽真空阀打开(步)
MOVF(469) D4176 D1362  ; #4电池真空压力表读数(实际真空值), 4#腔体充氦时电池实际压力（浮点）
LD TR0
@AND 13.06  ; #4腔体氦检阀
MOVF(469) D4070 D1364  ; 腔体4实际真空值(浮点), 4#腔体氦检时腔体实际压力（浮点）
LD TR0
AND 1487.01  ; 4#腔平移气缸后退(步)
MOVF(469) &0 D1362  ; 4#腔体充氦时电池实际压力（浮点）
MOVF(469) &0 D1364  ; 4#腔体氦检时腔体实际压力（浮点）

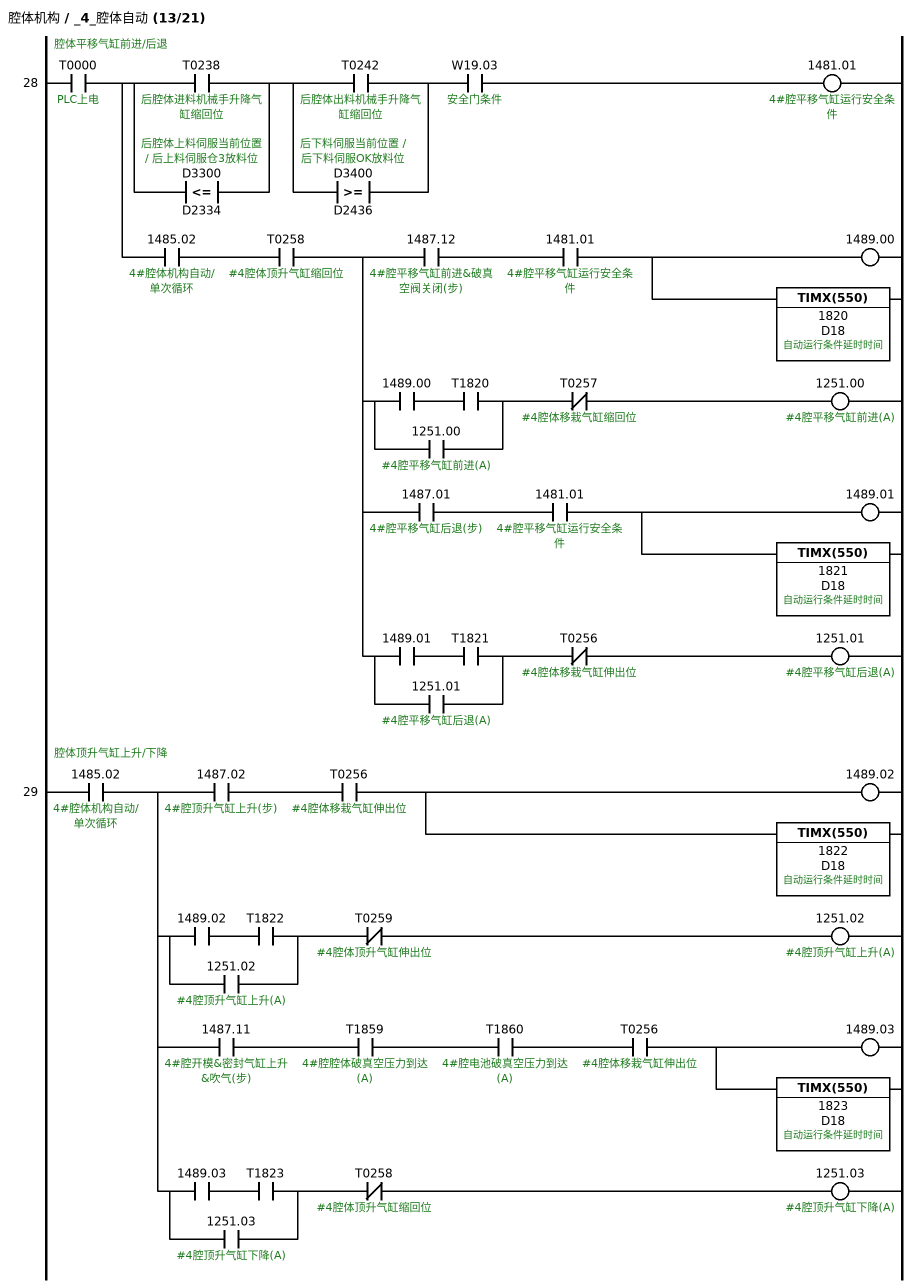
; rung 28: 腔体平移气缸前进/后退
LD T0000  ; PLC上电
OUT TR0
LD T0238  ; 后腔体进料机械手升降气缸缩回位
OR<=SL(318) D3300 D2334  ; 后腔体上料伺服当前位置, 后上料伺服仓3放料位
ANDLD
LD T0242  ; 后腔体出料机械手升降气缸缩回位
OR>=SL(328) D3400 D2436  ; 后下料伺服当前位置, 后下料伺服OK放料位
ANDLD
AND W19.03  ; 安全门条件
OUT 1481.01  ; 4#腔平移气缸运行安全条件
LD TR0
AND 1485.02  ; 4#腔体机构自动/单次循环
AND T0258  ; #4腔体顶升气缸缩回位
OUT TR0
AND 1487.12  ; 4#腔平移气缸前进&破真空阀关闭(步)
AND 1481.01  ; 4#腔平移气缸运行安全条件
OUT 1489.00
TIMX(550) 1820 D18  ; 自动运行条件延时时间
LD TR0
LD 1489.00
AND T1820
OR 1251.00  ; #4腔平移气缸前进(A)
ANDLD
ANDNOT T0257  ; #4腔体移栽气缸缩回位
OUT 1251.00  ; #4腔平移气缸前进(A)
LD TR0
AND 1487.01  ; 4#腔平移气缸后退(步)
AND 1481.01  ; 4#腔平移气缸运行安全条件
OUT 1489.01
TIMX(550) 1821 D18  ; 自动运行条件延时时间
LD TR0
LD 1489.01
AND T1821
OR 1251.01  ; #4腔平移气缸后退(A)
ANDLD
ANDNOT T0256  ; #4腔体移栽气缸伸出位
OUT 1251.01  ; #4腔平移气缸后退(A)
; rung 29: 腔体顶升气缸上升/下降
LD 1485.02  ; 4#腔体机构自动/单次循环
OUT TR0
AND 1487.02  ; 4#腔顶升气缸上升(步)
AND T0256  ; #4腔体移栽气缸伸出位
OUT 1489.02
TIMX(550) 1822 D18  ; 自动运行条件延时时间
LD TR0
LD 1489.02
AND T1822
OR 1251.02  ; #4腔顶升气缸上升(A)
ANDLD
ANDNOT T0259  ; #4腔体顶升气缸伸出位
OUT 1251.02  ; #4腔顶升气缸上升(A)
LD TR0
AND 1487.11  ; 4#腔开模&密封气缸上升&吹气(步)
AND T1859  ; 4#腔腔体破真空压力到达(A)
AND T1860  ; 4#腔电池破真空压力到达(A)
AND T0256  ; #4腔体移栽气缸伸出位
OUT 1489.03
TIMX(550) 1823 D18  ; 自动运行条件延时时间
LD TR0
LD 1489.03
AND T1823
OR 1251.03  ; #4腔顶升气缸下降(A)
ANDLD
ANDNOT T0258  ; #4腔体顶升气缸缩回位
OUT 1251.03  ; #4腔顶升气缸下降(A)

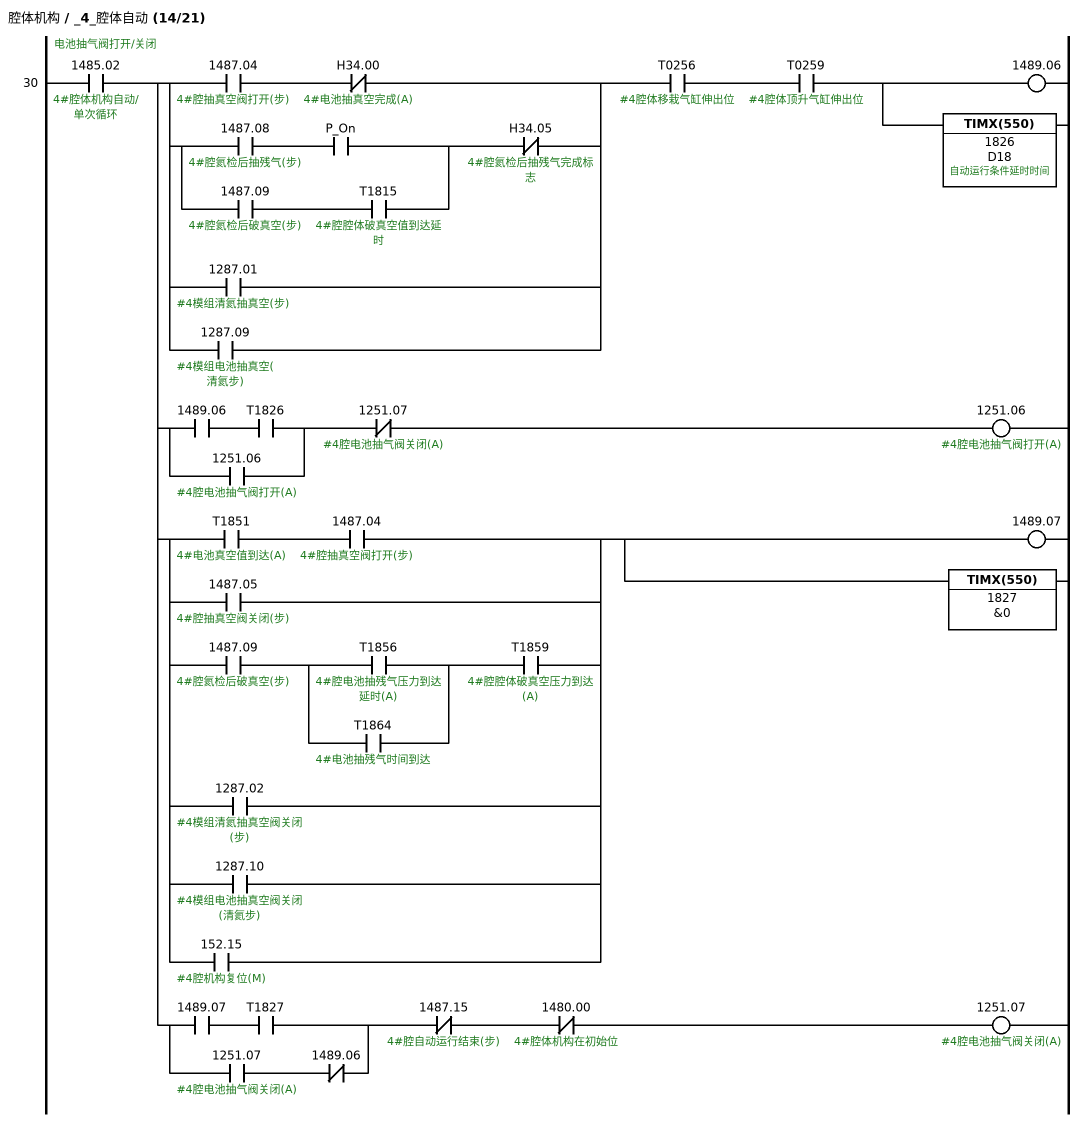
; rung 30: 电池抽气阀打开/关闭
LD 1485.02  ; 4#腔体机构自动/单次循环
OUT TR0
LD 1487.04  ; 4#腔抽真空阀打开(步)
ANDNOT H34.00  ; 4#电池抽真空完成(A)
LD 1487.08  ; 4#腔氦检后抽残气(步)
AND P_On
LD 1487.09  ; 4#腔氦检后破真空(步)
AND T1815  ; 4#腔腔体破真空值到达延时
ORLD
ANDNOT H34.05  ; 4#腔氦检后抽残气完成标志
ORLD
OR 1287.01  ; #4模组清氦抽真空(步)
OR 1287.09  ; #4模组电池抽真空(清氦步)
ANDLD
AND T0256  ; #4腔体移栽气缸伸出位
AND T0259  ; #4腔体顶升气缸伸出位
OUT 1489.06
TIMX(550) 1826 D18  ; 自动运行条件延时时间
LD TR0
LD 1489.06
AND T1826
OR 1251.06  ; #4腔电池抽气阀打开(A)
ANDLD
ANDNOT 1251.07  ; #4腔电池抽气阀关闭(A)
OUT 1251.06  ; #4腔电池抽气阀打开(A)
LD TR0
LD T1851  ; 4#电池真空值到达(A)
AND 1487.04  ; 4#腔抽真空阀打开(步)
OR 1487.05  ; 4#腔抽真空阀关闭(步)
LD 1487.09  ; 4#腔氦检后破真空(步)
LD T1856  ; 4#腔电池抽残气压力到达延时(A)
OR T1864  ; 4#电池抽残气时间到达
ANDLD
AND T1859  ; 4#腔腔体破真空压力到达(A)
ORLD
OR 1287.02  ; #4模组清氦抽真空阀关闭(步)
OR 1287.10  ; #4模组电池抽真空阀关闭(清氦步)
OR 152.15  ; #4腔机构复位(M)
ANDLD
OUT 1489.07
TIMX(550) 1827 &0
LD TR0
LD 1489.07
AND T1827
LD 1251.07  ; #4腔电池抽气阀关闭(A)
ANDNOT 1489.06
ORLD
ANDLD
ANDNOT 1487.15  ; 4#腔自动运行结束(步)
ANDNOT 1480.00  ; 4#腔体机构在初始位
OUT 1251.07  ; #4腔电池抽气阀关闭(A)

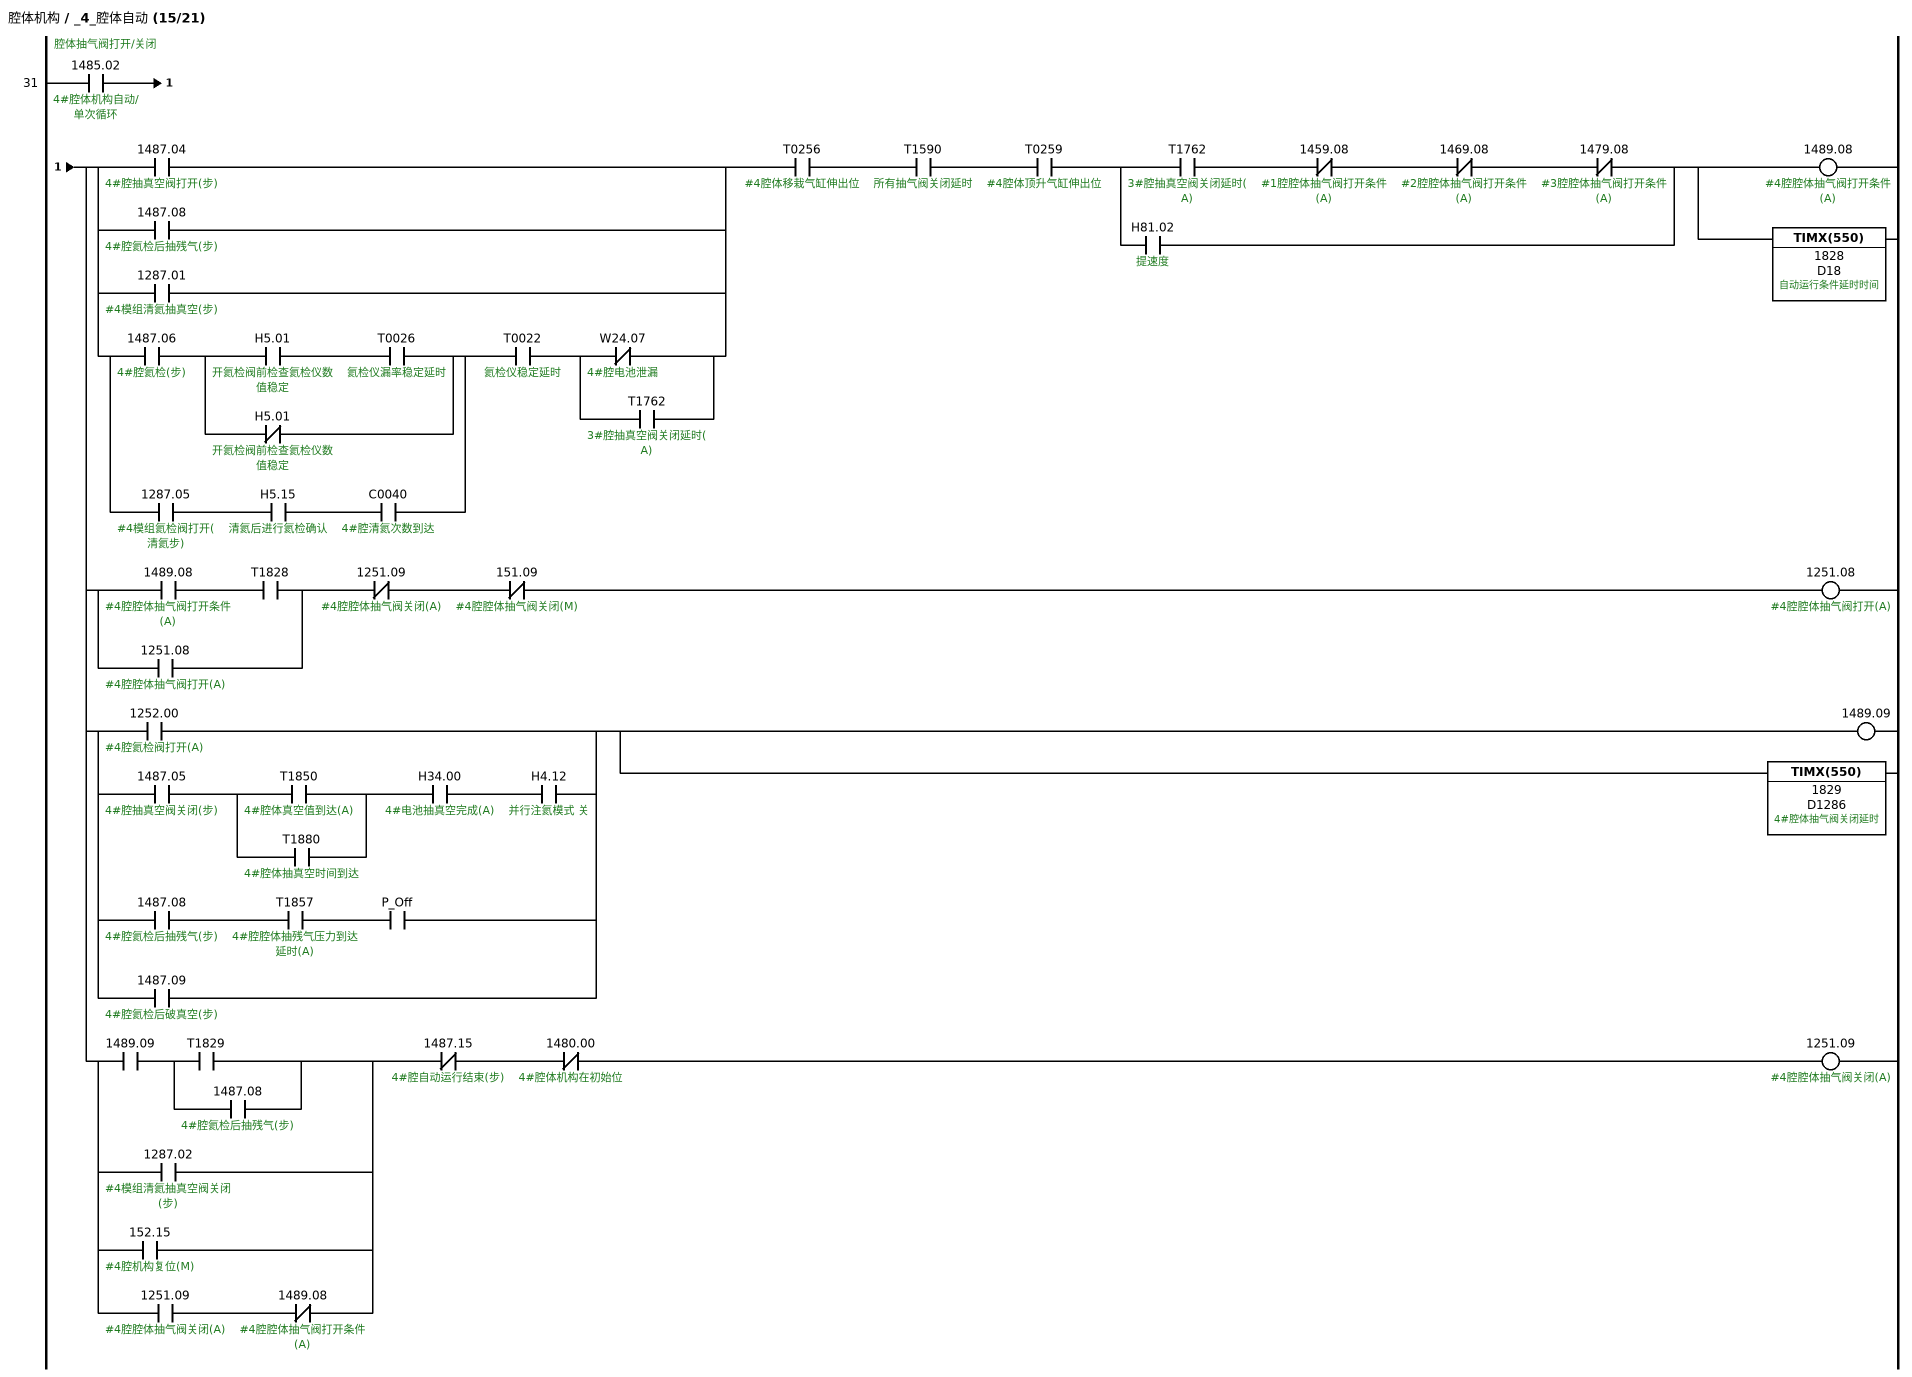
; rung 31: 腔体抽气阀打开/关闭
LD 1485.02  ; 4#腔体机构自动/单次循环
OUT TR0
LD 1487.04  ; 4#腔抽真空阀打开(步)
OR 1487.08  ; 4#腔氦检后抽残气(步)
OR 1287.01  ; #4模组清氦抽真空(步)
LD 1487.06  ; 4#腔氦检(步)
LD H5.01  ; 开氦检阀前检查氦检仪数值稳定
AND T0026  ; 氦检仪漏率稳定延时
ORNOT H5.01  ; 开氦检阀前检查氦检仪数值稳定
ANDLD
LD 1287.05  ; #4模组氦检阀打开(清氦步)
AND H5.15  ; 清氦后进行氦检确认
AND C0040  ; 4#腔清氦次数到达
ORLD
AND T0022  ; 氦检仪稳定延时
LDNOT W24.07  ; 4#腔电池泄漏
OR T1762  ; 3#腔抽真空阀关闭延时(A)
ANDLD
ORLD
ANDLD
AND T0256  ; #4腔体移栽气缸伸出位
AND T1590  ; 所有抽气阀关闭延时
AND T0259  ; #4腔体顶升气缸伸出位
LD T1762  ; 3#腔抽真空阀关闭延时(A)
ANDNOT 1459.08  ; #1腔腔体抽气阀打开条件(A)
ANDNOT 1469.08  ; #2腔腔体抽气阀打开条件(A)
ANDNOT 1479.08  ; #3腔腔体抽气阀打开条件(A)
OR H81.02  ; 提速度
ANDLD
OUT 1489.08  ; #4腔腔体抽气阀打开条件(A)
TIMX(550) 1828 D18  ; 自动运行条件延时时间
LD TR0
LD 1489.08  ; #4腔腔体抽气阀打开条件(A)
AND T1828
OR 1251.08  ; #4腔腔体抽气阀打开(A)
ANDLD
ANDNOT 1251.09  ; #4腔腔体抽气阀关闭(A)
ANDNOT 151.09  ; #4腔腔体抽气阀关闭(M)
OUT 1251.08  ; #4腔腔体抽气阀打开(A)
LD TR0
LD 1252.00  ; #4腔氦检阀打开(A)
LD 1487.05  ; 4#腔抽真空阀关闭(步)
LD T1850  ; 4#腔体真空值到达(A)
OR T1880  ; 4#腔体抽真空时间到达
ANDLD
AND H34.00  ; 4#电池抽真空完成(A)
AND H4.12  ; 并行注氦模式 关
ORLD
LD 1487.08  ; 4#腔氦检后抽残气(步)
AND T1857  ; 4#腔腔体抽残气压力到达延时(A)
AND P_Off
ORLD
OR 1487.09  ; 4#腔氦检后破真空(步)
ANDLD
OUT 1489.09
TIMX(550) 1829 D1286  ; 4#腔体抽气阀关闭延时
LD TR0
LD 1489.09
LD T1829
OR 1487.08  ; 4#腔氦检后抽残气(步)
ANDLD
OR 1287.02  ; #4模组清氦抽真空阀关闭(步)
OR 152.15  ; #4腔机构复位(M)
LD 1251.09  ; #4腔腔体抽气阀关闭(A)
ANDNOT 1489.08  ; #4腔腔体抽气阀打开条件(A)
ORLD
ANDLD
ANDNOT 1487.15  ; 4#腔自动运行结束(步)
ANDNOT 1480.00  ; 4#腔体机构在初始位
OUT 1251.09  ; #4腔腔体抽气阀关闭(A)

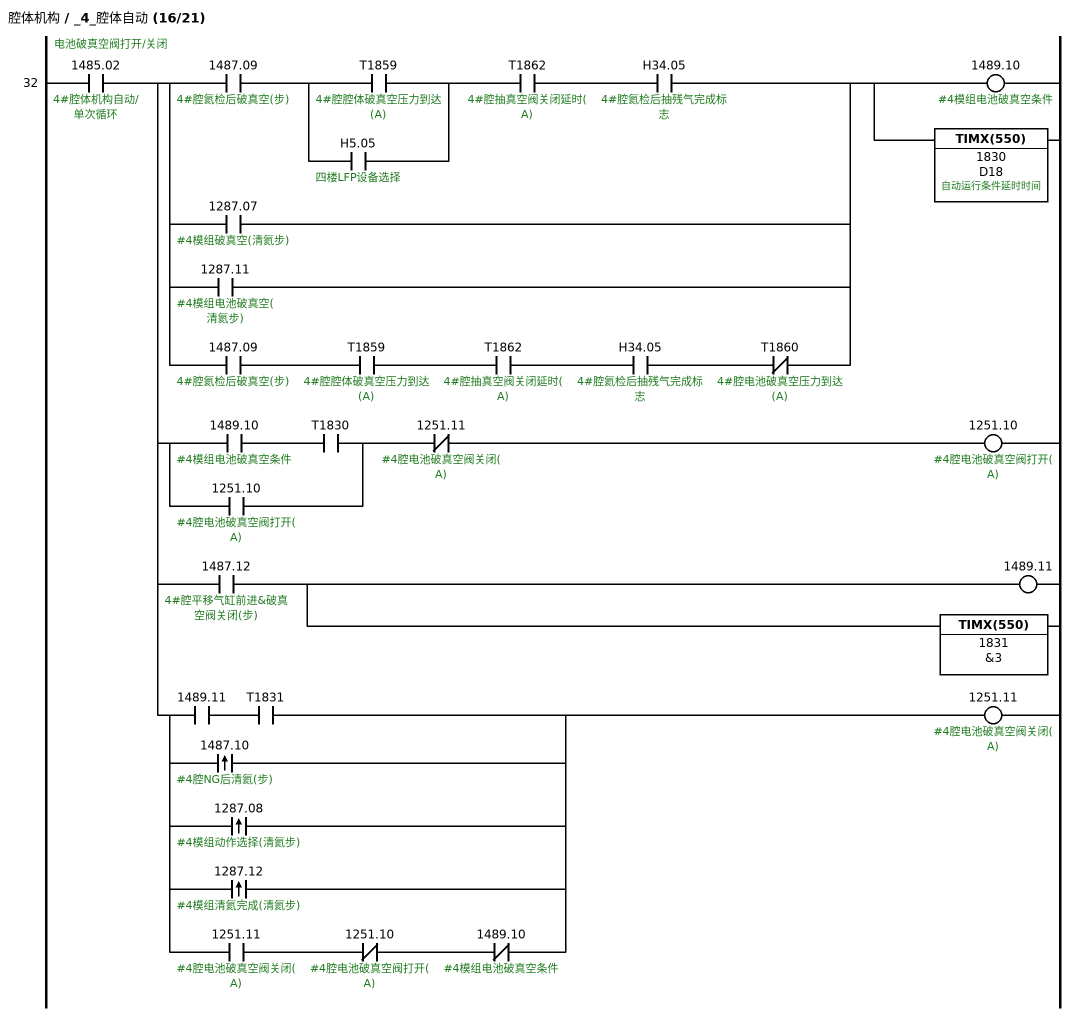
; rung 32: 电池破真空阀打开/关闭
LD 1485.02  ; 4#腔体机构自动/单次循环
OUT TR0
LD 1487.09  ; 4#腔氦检后破真空(步)
LD T1859  ; 4#腔腔体破真空压力到达(A)
OR H5.05  ; 四楼LFP设备选择
ANDLD
AND T1862  ; 4#腔抽真空阀关闭延时(A)
AND H34.05  ; 4#腔氦检后抽残气完成标志
OR 1287.07  ; #4模组破真空(清氦步)
OR 1287.11  ; #4模组电池破真空(清氦步)
LD 1487.09  ; 4#腔氦检后破真空(步)
AND T1859  ; 4#腔腔体破真空压力到达(A)
AND T1862  ; 4#腔抽真空阀关闭延时(A)
AND H34.05  ; 4#腔氦检后抽残气完成标志
ANDNOT T1860  ; 4#腔电池破真空压力到达(A)
ORLD
ANDLD
OUT 1489.10  ; #4模组电池破真空条件
TIMX(550) 1830 D18  ; 自动运行条件延时时间
LD TR0
LD 1489.10  ; #4模组电池破真空条件
AND T1830
OR 1251.10  ; #4腔电池破真空阀打开(A)
ANDLD
ANDNOT 1251.11  ; #4腔电池破真空阀关闭(A)
OUT 1251.10  ; #4腔电池破真空阀打开(A)
LD TR0
AND 1487.12  ; 4#腔平移气缸前进&破真空阀关闭(步)
OUT 1489.11
TIMX(550) 1831 &3
LD TR0
LD 1489.11
AND T1831
@OR 1487.10  ; #4腔NG后清氦(步)
@OR 1287.08  ; #4模组动作选择(清氦步)
@OR 1287.12  ; #4模组清氦完成(清氦步)
LD 1251.11  ; #4腔电池破真空阀关闭(A)
ANDNOT 1251.10  ; #4腔电池破真空阀打开(A)
ANDNOT 1489.10  ; #4模组电池破真空条件
ORLD
ANDLD
OUT 1251.11  ; #4腔电池破真空阀关闭(A)

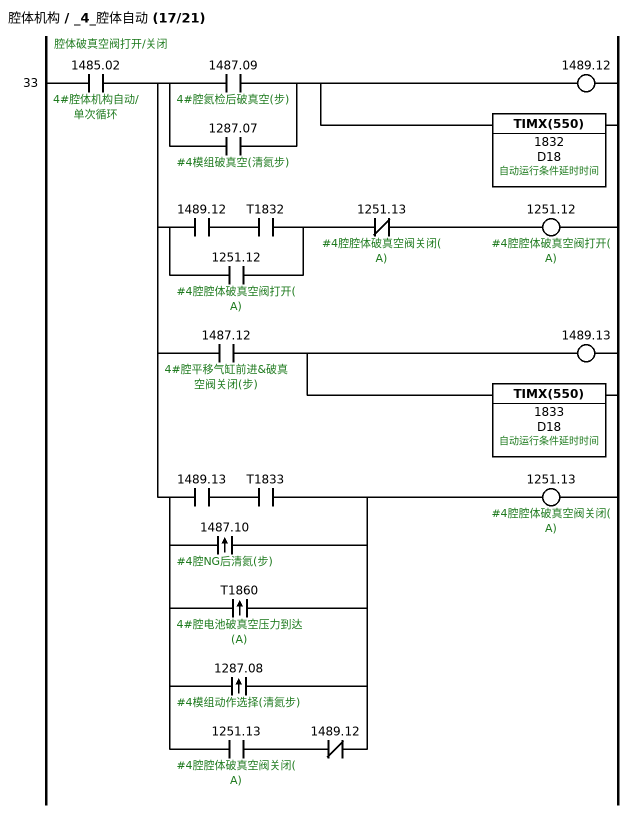
; rung 33: 腔体破真空阀打开/关闭
LD 1485.02  ; 4#腔体机构自动/单次循环
OUT TR0
LD 1487.09  ; 4#腔氦检后破真空(步)
OR 1287.07  ; #4模组破真空(清氦步)
ANDLD
OUT 1489.12
TIMX(550) 1832 D18  ; 自动运行条件延时时间
LD TR0
LD 1489.12
AND T1832
OR 1251.12  ; #4腔腔体破真空阀打开(A)
ANDLD
ANDNOT 1251.13  ; #4腔腔体破真空阀关闭(A)
OUT 1251.12  ; #4腔腔体破真空阀打开(A)
LD TR0
AND 1487.12  ; 4#腔平移气缸前进&破真空阀关闭(步)
OUT 1489.13
TIMX(550) 1833 D18  ; 自动运行条件延时时间
LD TR0
LD 1489.13
AND T1833
@OR 1487.10  ; #4腔NG后清氦(步)
@OR T1860  ; 4#腔电池破真空压力到达(A)
@OR 1287.08  ; #4模组动作选择(清氦步)
LD 1251.13  ; #4腔腔体破真空阀关闭(A)
ANDNOT 1489.12
ORLD
ANDLD
OUT 1251.13  ; #4腔腔体破真空阀关闭(A)

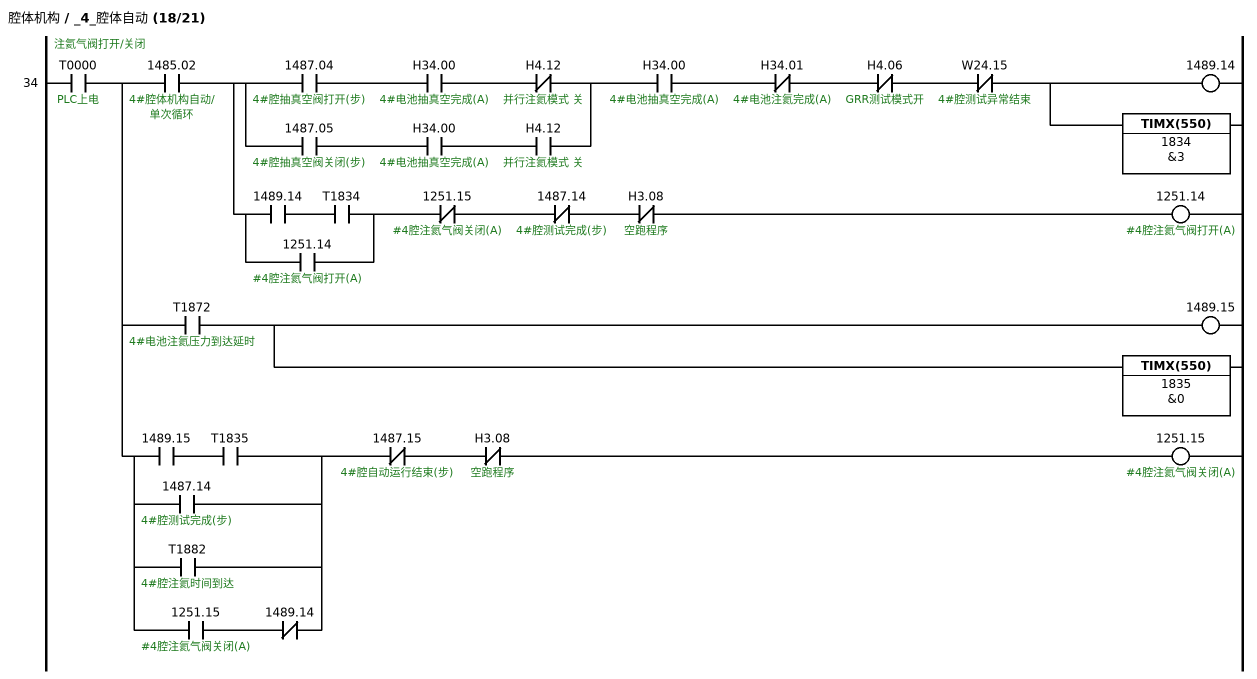
; rung 34: 注氦气阀打开/关闭
LD T0000  ; PLC上电
OUT TR0
AND 1485.02  ; 4#腔体机构自动/单次循环
OUT TR1
LD 1487.04  ; 4#腔抽真空阀打开(步)
AND H34.00  ; 4#电池抽真空完成(A)
ANDNOT H4.12  ; 并行注氦模式 关
LD 1487.05  ; 4#腔抽真空阀关闭(步)
AND H34.00  ; 4#电池抽真空完成(A)
AND H4.12  ; 并行注氦模式 关
ORLD
ANDLD
AND H34.00  ; 4#电池抽真空完成(A)
ANDNOT H34.01  ; 4#电池注氦完成(A)
ANDNOT H4.06  ; GRR测试模式开
ANDNOT W24.15  ; 4#腔测试异常结束
OUT 1489.14
TIMX(550) 1834 &3
LD TR1
LD 1489.14
AND T1834
OR 1251.14  ; #4腔注氦气阀打开(A)
ANDLD
ANDNOT 1251.15  ; #4腔注氦气阀关闭(A)
ANDNOT 1487.14  ; 4#腔测试完成(步)
ANDNOT H3.08  ; 空跑程序
OUT 1251.14  ; #4腔注氦气阀打开(A)
LD TR0
AND T1872  ; 4#电池注氦压力到达延时
OUT 1489.15
TIMX(550) 1835 &0
LD TR0
LD 1489.15
AND T1835
OR 1487.14  ; 4#腔测试完成(步)
OR T1882  ; 4#腔注氦时间到达
LD 1251.15  ; #4腔注氦气阀关闭(A)
ANDNOT 1489.14
ORLD
ANDLD
ANDNOT 1487.15  ; 4#腔自动运行结束(步)
ANDNOT H3.08  ; 空跑程序
OUT 1251.15  ; #4腔注氦气阀关闭(A)

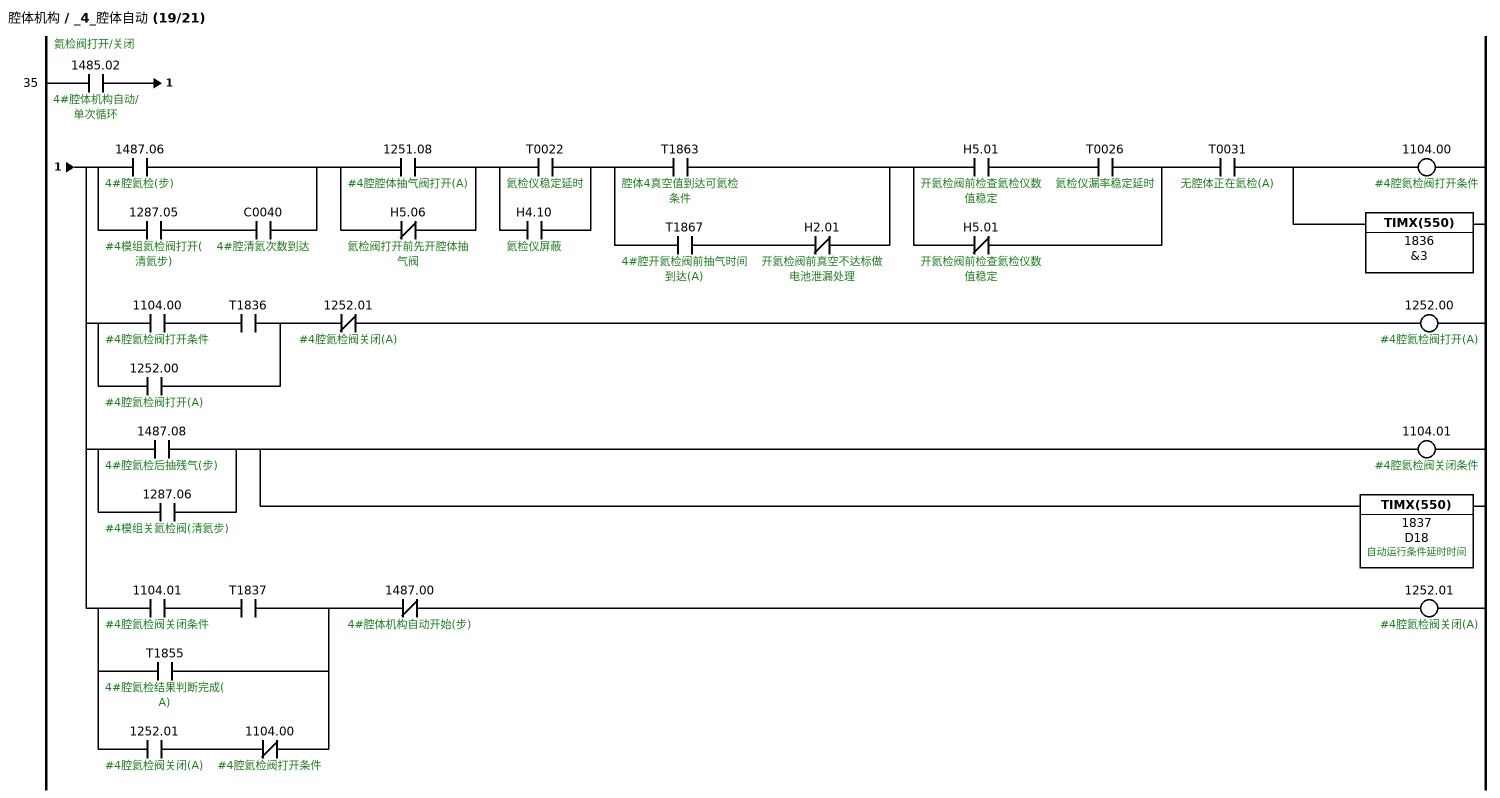
; rung 35: 氦检阀打开/关闭
LD 1485.02  ; 4#腔体机构自动/单次循环
OUT TR0
LD 1487.06  ; 4#腔氦检(步)
LD 1287.05  ; #4模组氦检阀打开(清氦步)
AND C0040  ; 4#腔清氦次数到达
ORLD
ANDLD
LD 1251.08  ; #4腔腔体抽气阀打开(A)
ORNOT H5.06  ; 氦检阀打开前先开腔体抽气阀
ANDLD
LD T0022  ; 氦检仪稳定延时
OR H4.10  ; 氦检仪屏蔽
ANDLD
LD T1863  ; 腔体4真空值到达可氦检条件
LD T1867  ; 4#腔开氦检阀前抽气时间到达(A)
ANDNOT H2.01  ; 开氦检阀前真空不达标做电池泄漏处理
ORLD
ANDLD
LD H5.01  ; 开氦检阀前检查氦检仪数值稳定
AND T0026  ; 氦检仪漏率稳定延时
ORNOT H5.01  ; 开氦检阀前检查氦检仪数值稳定
ANDLD
AND T0031  ; 无腔体正在氦检(A)
OUT 1104.00  ; #4腔氦检阀打开条件
TIMX(550) 1836 &3
LD TR0
LD 1104.00  ; #4腔氦检阀打开条件
AND T1836
OR 1252.00  ; #4腔氦检阀打开(A)
ANDLD
ANDNOT 1252.01  ; #4腔氦检阀关闭(A)
OUT 1252.00  ; #4腔氦检阀打开(A)
LD TR0
LD 1487.08  ; 4#腔氦检后抽残气(步)
OR 1287.06  ; #4模组关氦检阀(清氦步)
ANDLD
OUT 1104.01  ; #4腔氦检阀关闭条件
TIMX(550) 1837 D18  ; 自动运行条件延时时间
LD TR0
LD 1104.01  ; #4腔氦检阀关闭条件
AND T1837
OR T1855  ; 4#腔氦检结果判断完成(A)
LD 1252.01  ; #4腔氦检阀关闭(A)
ANDNOT 1104.00  ; #4腔氦检阀打开条件
ORLD
ANDLD
ANDNOT 1487.00  ; 4#腔体机构自动开始(步)
OUT 1252.01  ; #4腔氦检阀关闭(A)

